C05450=1130.712,124.899,-57.710,-179.760,8.342,149.534
C05451=1130.717,124.650,-57.689,-179.762,8.338,149.533
C05452=1130.723,124.401,-57.670,-179.763,8.335,149.533
C05453=1130.727,124.152,-57.649,-179.765,8.332,149.533
C05454=1130.732,123.903,-57.630,-179.768,8.328,149.533
C05455=1130.736,123.654,-57.609,-179.770,8.325,149.532
C05456=1130.741,123.404,-57.589,-179.771,8.321,149.532
C05457=1130.746,123.156,-57.569,-179.773,8.318,149.532
C05458=1130.751,122.906,-57.550,-179.775,8.314,149.531
C05459=1130.756,122.657,-57.530,-179.777,8.311,149.531
C05460=1130.760,122.408,-57.510,-179.778,8.308,149.531
C05461=1130.765,122.159,-57.491,-179.780,8.304,149.531
C05462=1130.770,121.910,-57.470,-179.782,8.301,149.530
C05463=1130.775,121.660,-57.450,-179.784,8.297,149.530
C05464=1130.779,121.411,-57.431,-179.786,8.294,149.530
C05465=1130.784,121.162,-57.411,-179.788,8.291,149.530
C05466=1130.789,120.913,-57.391,-179.789,8.287,149.529
C05467=1130.794,120.663,-57.371,-179.791,8.284,149.529
C05468=1130.798,120.414,-57.351,-179.793,8.280,149.529
C05469=1130.804,120.166,-57.332,-179.795,8.278,149.529
C05470=1130.808,119.916,-57.312,-179.797,8.274,149.528
C05471=1130.813,119.667,-57.292,-179.799,8.271,149.528
C05472=1130.818,119.417,-57.272,-179.800,8.267,149.528
C05473=1130.823,119.169,-57.253,-179.803,8.263,149.528
C05474=1130.827,118.920,-57.233,-179.805,8.260,149.527
C05475=1130.831,118.670,-57.213,-179.806,8.257,149.527
C05476=1130.837,118.422,-57.194,-179.808,8.254,149.527
C05477=1130.841,118.172,-57.174,-179.810,8.250,149.526
C05478=1130.846,117.922,-57.155,-179.812,8.246,149.526
C05479=1130.851,117.674,-57.135,-179.814,8.243,149.526
C05480=1130.855,117.459,-57.118,-179.815,8.240,149.526
C05481=1130.859,117.244,-57.101,-179.817,8.236,149.526
C05482=1130.864,117.029,-57.084,-179.819,8.234,149.525
C05483=1130.868,116.814,-57.067,-179.820,8.231,149.525
C05484=1130.872,116.599,-57.051,-179.822,8.227,149.525
C05485=1130.877,116.384,-57.034,-179.824,8.225,149.525
C05486=1130.880,116.169,-57.017,-179.825,8.222,149.524
C05487=1130.884,115.954,-57.000,-179.827,8.219,149.524
C05488=1130.889,115.705,-56.981,-179.829,8.215,149.524
C05489=1130.894,115.456,-56.961,-179.831,8.212,149.524
C05490=1130.898,115.207,-56.941,-179.832,8.208,149.523
C05491=1130.904,114.958,-56.922,-179.834,8.205,149.523
C05492=1130.908,114.709,-56.903,-179.837,8.201,149.523
C05493=1130.913,114.460,-56.883,-179.839,8.198,149.523
C05494=1130.918,114.210,-56.864,-179.841,8.194,149.522
C05495=1130.922,113.961,-56.844,-179.843,8.191,149.522
C05496=1130.928,113.712,-56.825,-179.844,8.187,149.522
C05497=1130.932,113.463,-56.806,-179.846,8.184,149.522
C05498=1130.937,113.214,-56.786,-179.848,8.180,149.521
C05499=1130.942,112.964,-56.767,-179.851,8.177,149.521
C05500=1130.947,112.715,-56.748,-179.853,8.173,149.521
C05501=1130.951,112.466,-56.728,-179.854,8.169,149.521
C05502=1130.956,112.216,-56.709,-179.856,8.166,149.520
C05503=1130.962,111.967,-56.690,-179.858,8.162,149.520
C05504=1130.966,111.718,-56.671,-179.860,8.159,149.520
C05505=1130.971,111.469,-56.652,-179.862,8.155,149.520
C05506=1130.976,111.219,-56.632,-179.864,8.152,149.519
C05507=1130.980,110.971,-56.614,-179.866,8.148,149.519
C05508=1130.985,110.721,-56.594,-179.868,8.144,149.519
C05509=1130.990,110.472,-56.575,-179.871,8.140,149.519
C05510=1130.994,110.223,-56.556,-179.874,8.136,149.519
C05511=1131.000,109.974,-56.537,-179.877,8.132,149.518
C05512=1131.005,109.724,-56.517,-179.879,8.128,149.518
C05513=1131.009,109.475,-56.499,-179.881,8.124,149.518
C05514=1131.014,109.226,-56.479,-179.884,8.120,149.518
C05515=1131.019,108.977,-56.460,-179.887,8.117,149.518
C05516=1131.024,108.727,-56.441,-179.889,8.112,149.517
C05517=1131.029,108.478,-56.422,-179.892,8.108,149.517
C05518=1131.033,108.229,-56.403,-179.894,8.105,149.517
C05519=1131.038,107.980,-56.384,-179.897,8.100,149.517
C05520=1131.043,107.730,-56.365,-179.899,8.096,149.517
C05521=1131.048,107.481,-56.346,-179.901,8.093,149.516
C05522=1131.052,107.232,-56.327,-179.904,8.088,149.516
C05523=1131.058,106.983,-56.308,-179.907,8.084,149.516
C05524=1131.062,106.734,-56.290,-179.909,8.081,149.516
C05525=1131.067,106.484,-56.271,-179.912,8.076,149.515
C05526=1131.072,106.235,-56.252,-179.914,8.072,149.515
C05527=1131.077,105.986,-56.232,-179.916,8.068,149.515
C05528=1131.082,105.737,-56.214,-179.919,8.064,149.515
C05529=1131.086,105.487,-56.195,-179.921,8.060,149.514
C05530=1131.091,105.238,-56.177,-179.923,8.056,149.514
C05531=1131.096,104.989,-56.158,-179.925,8.052,149.514
C05532=1131.101,104.739,-56.139,-179.928,8.048,149.514
C05533=1131.106,104.491,-56.120,-179.931,8.044,149.514
C05534=1131.111,104.241,-56.102,-179.932,8.040,149.513
C05535=1131.115,103.992,-56.083,-179.935,8.036,149.513
C05536=1131.120,103.777,-56.067,-179.936,8.033,149.513
C05537=1131.123,103.562,-56.050,-179.939,8.030,149.512
C05538=1131.128,103.347,-56.034,-179.941,8.026,149.512
C05539=1131.132,103.132,-56.019,-179.943,8.023,149.512
C05540=1131.136,102.917,-56.002,-179.944,8.019,149.512
C05541=1131.140,102.702,-55.987,-179.946,8.015,149.511
C05542=1131.145,102.487,-55.970,-179.948,8.012,149.511
C05543=1131.149,102.272,-55.955,-179.950,8.008,149.511
C05544=1131.154,102.023,-55.936,-179.952,8.005,149.511
C05545=1131.158,101.773,-55.917,-179.955,8.000,149.510
C05546=1131.163,101.525,-55.898,-179.957,7.996,149.510
C05547=1131.169,101.275,-55.880,-179.958,7.993,149.510
C05548=1131.173,101.025,-55.862,-179.961,7.988,149.509
C05549=1131.178,100.776,-55.844,-179.963,7.984,149.509
C05550=1131.183,100.527,-55.825,-179.965,7.980,149.509
C05551=1131.188,100.278,-55.806,-179.967,7.976,149.508
C05552=1131.193,100.028,-55.788,-179.969,7.973,149.508
C05553=1131.197,99.780,-55.769,-179.971,7.968,149.508
C05554=1131.202,99.530,-55.751,-179.973,7.965,149.508
C05555=1131.208,99.281,-55.733,-179.976,7.960,149.507
C05556=1131.212,99.031,-55.714,-179.978,7.956,149.507
C05557=1131.217,98.782,-55.696,-179.979,7.953,149.506
C05558=1131.222,98.533,-55.678,-179.981,7.948,149.506
C05559=1131.226,98.284,-55.660,-179.983,7.944,149.506
C05560=1131.231,98.034,-55.641,-179.985,7.940,149.505
C05561=1131.236,97.785,-55.623,-179.987,7.936,149.505
C05562=1131.241,97.536,-55.605,-179.989,7.932,149.505
C05563=1131.246,97.286,-55.587,-179.991,7.928,149.504
C05564=1131.251,97.038,-55.568,-179.993,7.925,149.504
C05565=1131.255,96.788,-55.550,-179.995,7.920,149.504
C05566=1131.261,96.538,-55.531,-179.997,7.916,149.503
C05567=1131.266,96.289,-55.513,-179.998,7.912,149.503
C05568=1131.271,96.040,-55.495,180.000,7.909,149.502
C05569=1131.276,95.791,-55.477,179.997,7.904,149.502
C05570=1131.280,95.542,-55.459,179.996,7.900,149.502
C05571=1131.285,95.292,-55.441,179.994,7.896,149.501
C05572=1131.290,95.043,-55.423,179.992,7.893,149.501
C05573=1131.295,94.794,-55.405,179.990,7.888,149.500
C05574=1131.299,94.544,-55.387,179.989,7.884,149.500
C05575=1131.304,94.295,-55.369,179.987,7.881,149.500
C05576=1131.309,94.046,-55.351,179.985,7.877,149.499
C05577=1131.315,93.797,-55.332,179.983,7.873,149.499
C05578=1131.319,93.547,-55.314,179.982,7.869,149.499
C05579=1131.324,93.297,-55.296,179.980,7.864,149.498
C05580=1131.329,93.048,-55.278,179.978,7.860,149.498
C05581=1131.334,92.799,-55.260,179.976,7.856,149.497
C05582=1131.339,92.550,-55.242,179.975,7.853,149.497
C05583=1131.344,92.301,-55.224,179.973,7.849,149.496
C05584=1131.349,92.051,-55.207,179.972,7.845,149.496
C05585=1131.354,91.802,-55.189,179.970,7.841,149.496
C05586=1131.359,91.553,-55.171,179.968,7.837,149.495
C05587=1131.364,91.303,-55.153,179.967,7.833,149.495
C05588=1131.368,91.055,-55.136,179.965,7.829,149.494
C05589=1131.372,90.805,-55.117,179.964,7.825,149.494
C05590=1131.377,90.555,-55.100,179.962,7.821,149.493
C05591=1131.382,90.306,-55.082,179.960,7.817,149.493
C05592=1131.387,90.032,-55.062,179.958,7.813,149.493
C05593=1131.393,89.758,-55.043,179.957,7.809,149.492
C05594=1131.418,88.513,-54.953,-179.494,6.756,149.096
C05595=1131.423,88.264,-54.935,-179.496,6.755,149.097
C05596=1131.428,88.015,-54.918,-179.499,6.754,149.097
C05597=1131.433,87.767,-54.901,-179.502,6.753,149.098
C05598=1131.437,87.518,-54.883,-179.505,6.751,149.098
C05599=1131.443,87.268,-54.866,-179.508,6.749,149.099
C05600=1131.448,87.019,-54.848,-179.510,6.748,149.099
C05601=1131.453,86.769,-54.831,-179.513,6.746,149.100
C05602=1131.457,86.520,-54.814,-179.516,6.744,149.100
C05603=1131.462,86.271,-54.796,-179.518,6.744,149.101
C05604=1131.467,86.021,-54.778,-179.521,6.742,149.101
C05605=1131.472,85.772,-54.761,-179.524,6.740,149.101
C05606=1131.476,85.523,-54.744,-179.527,6.739,149.102
C05607=1131.482,85.273,-54.726,-179.529,6.737,149.102
C05608=1131.487,85.024,-54.708,-179.532,6.735,149.103
C05609=1131.492,84.775,-54.692,-179.535,6.734,149.103
C05610=1131.497,84.526,-54.674,-179.538,6.733,149.104
C05611=1131.502,84.276,-54.657,-179.540,6.732,149.104
C05612=1131.506,84.027,-54.640,-179.543,6.730,149.105
C05613=1131.511,83.777,-54.622,-179.546,6.728,149.105
C05614=1131.516,83.528,-54.605,-179.548,6.727,149.106
C05615=1131.521,83.278,-54.588,-179.551,6.725,149.106
C05616=1131.526,83.029,-54.570,-179.554,6.724,149.107
C05617=1131.532,82.780,-54.553,-179.557,6.723,149.107
C05618=1131.536,82.531,-54.536,-179.559,6.721,149.107
C05619=1131.541,82.281,-54.519,-179.562,6.720,149.108
C05620=1131.545,82.032,-54.502,-179.565,6.718,149.108
C05621=1131.550,81.783,-54.484,-179.568,6.716,149.109
C05622=1131.556,81.533,-54.467,-179.571,6.715,149.109
C05623=1131.561,81.284,-54.451,-179.573,6.714,149.110
C05624=1131.566,81.034,-54.433,-179.576,6.713,149.110
C05625=1131.570,80.785,-54.416,-179.578,6.711,149.111
C05626=1131.575,80.536,-54.399,-179.581,6.709,149.111
C05627=1131.580,80.286,-54.382,-179.584,6.708,149.112
C05628=1131.586,80.037,-54.365,-179.587,6.706,149.112
C05629=1131.591,79.788,-54.347,-179.589,6.705,149.113
C05630=1131.595,79.519,-54.329,-179.592,6.704,149.113
C05631=1131.601,79.251,-54.311,-179.595,6.703,149.114
C05632=1131.606,78.982,-54.293,-179.599,6.700,149.114
C05633=1131.611,78.714,-54.274,-179.601,6.698,149.115
C05634=1131.616,78.465,-54.258,-179.604,6.698,149.115
C05635=1131.621,78.215,-54.240,-179.607,6.696,149.116
C05636=1131.626,77.966,-54.224,-179.610,6.695,149.116
C05637=1131.631,77.716,-54.206,-179.612,6.693,149.116
C05638=1131.636,77.468,-54.189,-179.615,6.691,149.117
C05639=1131.641,77.218,-54.172,-179.617,6.691,149.117
C05640=1131.646,76.968,-54.155,-179.620,6.689,149.118
C05641=1131.651,76.718,-54.138,-179.623,6.688,149.118
C05642=1131.656,76.470,-54.122,-179.626,6.686,149.119
C05643=1131.661,76.220,-54.105,-179.629,6.684,149.119
C05644=1131.666,75.970,-54.088,-179.631,6.683,149.120
C05645=1131.671,75.721,-54.071,-179.634,6.682,149.120
C05646=1131.676,75.472,-54.054,-179.637,6.681,149.121
C05647=1131.680,75.222,-54.038,-179.640,6.679,149.121
C05648=1131.686,74.973,-54.020,-179.642,6.678,149.122
C05649=1131.691,74.724,-54.004,-179.644,6.676,149.122
C05650=1131.696,74.474,-53.987,-179.648,6.675,149.123
C05651=1131.700,74.225,-53.970,-179.650,6.673,149.123
C05652=1131.706,73.976,-53.954,-179.653,6.672,149.124
C05653=1131.711,73.726,-53.937,-179.655,6.671,149.124
C05654=1131.715,73.476,-53.920,-179.658,6.669,149.125
C05655=1131.720,73.228,-53.904,-179.661,6.668,149.125
C05656=1131.726,72.978,-53.886,-179.664,6.666,149.126
C05657=1131.730,72.728,-53.870,-179.666,6.666,149.126
C05658=1131.735,72.480,-53.853,-179.669,6.664,149.126
C05659=1131.740,72.230,-53.836,-179.672,6.662,149.127
C05660=1131.745,71.980,-53.819,-179.675,6.661,149.128
C05661=1131.750,71.732,-53.803,-179.678,6.659,149.128
C05662=1131.755,71.482,-53.786,-179.680,6.659,149.128
C05663=1131.760,71.232,-53.769,-179.683,6.657,149.129
C05664=1131.765,70.983,-53.754,-179.685,6.655,149.129
C05665=1131.770,70.733,-53.736,-179.689,6.654,149.130
C05666=1131.775,70.484,-53.720,-179.691,6.653,149.130
C05667=1131.780,70.235,-53.703,-179.694,6.651,149.131
C05668=1131.784,69.985,-53.687,-179.696,6.650,149.131
C05669=1131.790,69.736,-53.670,-179.699,6.648,149.132
C05670=1131.795,69.486,-53.654,-179.702,6.648,149.132
C05671=1131.800,69.237,-53.638,-179.704,6.646,149.133
C05672=1131.804,68.988,-53.621,-179.707,6.644,149.133
C05673=1131.810,68.738,-53.604,-179.709,6.644,149.134
C05674=1131.815,68.489,-53.588,-179.713,6.642,149.134
C05675=1131.819,68.239,-53.571,-179.715,6.641,149.135
C05676=1131.825,67.990,-53.555,-179.718,6.639,149.135
C05677=1131.829,67.741,-53.538,-179.720,6.638,149.136
C05678=1131.835,67.491,-53.522,-179.723,6.637,149.136
C05679=1131.840,67.242,-53.506,-179.726,6.635,149.137
C05680=1131.844,66.992,-53.489,-179.729,6.634,149.137
C05681=1131.849,66.743,-53.473,-179.731,6.633,149.138
C05682=1131.854,66.493,-53.457,-179.734,6.631,149.138
C05683=1131.859,66.245,-53.440,-179.737,6.630,149.139
C05684=1131.864,65.994,-53.424,-179.739,6.629,149.139
C05685=1131.870,65.745,-53.407,-179.742,6.627,149.140
C05686=1131.874,65.496,-53.391,-179.745,6.626,149.140
C05687=1131.880,65.246,-53.375,-179.748,6.624,149.140
C05688=1131.884,64.997,-53.359,-179.750,6.624,149.141
C05689=1131.889,64.748,-53.342,-179.753,6.622,149.142
C05690=1131.894,64.498,-53.326,-179.756,6.620,149.142
C05691=1131.899,64.249,-53.310,-179.758,6.620,149.142
C05692=1131.904,63.999,-53.294,-179.761,6.618,149.143
C05693=1131.909,63.750,-53.278,-179.764,6.617,149.143
C05694=1131.914,63.500,-53.261,-179.767,6.615,149.144
C05695=1131.919,63.251,-53.245,-179.769,6.614,149.144
C05696=1131.924,63.002,-53.228,-179.772,6.613,149.145
C05697=1131.929,62.752,-53.213,-179.775,6.611,149.145
C05698=1131.934,62.503,-53.196,-179.777,6.610,149.146
C05699=1131.939,62.253,-53.180,-179.780,6.609,149.146
C05700=1131.944,62.004,-53.164,-179.783,6.607,149.147
C05701=1131.949,61.755,-53.148,-179.785,6.607,149.147
C05702=1131.953,61.505,-53.131,-179.788,6.605,149.148
C05703=1131.959,61.256,-53.116,-179.791,6.603,149.148
C05704=1131.964,61.006,-53.100,-179.793,6.603,149.149
C05705=1131.969,60.757,-53.084,-179.796,6.601,149.149
C05706=1131.974,60.507,-53.068,-179.799,6.600,149.150
C05707=1131.979,60.258,-53.051,-179.801,6.599,149.150
C05708=1131.984,60.009,-53.036,-179.804,6.598,149.151
C05709=1131.988,59.759,-53.019,-179.807,6.596,149.151
C05710=1131.994,59.510,-53.003,-179.809,6.595,149.152
C05711=1131.999,59.260,-52.988,-179.812,6.593,149.152
C05712=1132.004,59.011,-52.971,-179.815,6.592,149.153
C05713=1132.009,58.761,-52.956,-179.817,6.591,149.153
C05714=1132.014,58.511,-52.940,-179.820,6.590,149.154
C05715=1132.018,58.263,-52.924,-179.823,6.588,149.154
C05716=1132.024,58.013,-52.908,-179.825,6.588,149.155
C05717=1132.028,57.763,-52.892,-179.828,6.586,149.155
C05718=1132.034,57.514,-52.876,-179.831,6.584,149.156
C05719=1132.038,57.264,-52.860,-179.833,6.583,149.156
C05720=1132.044,57.015,-52.845,-179.836,6.582,149.157
C05721=1132.049,56.766,-52.828,-179.839,6.581,149.157
C05722=1132.054,56.516,-52.812,-179.841,6.580,149.158
C05723=1132.059,56.267,-52.797,-179.844,6.578,149.158
C05724=1132.064,56.017,-52.781,-179.847,6.577,149.159
C05725=1132.068,55.768,-52.765,-179.849,6.576,149.159
C05726=1132.073,55.519,-52.749,-179.852,6.574,149.160
C05727=1132.079,55.269,-52.734,-179.854,6.574,149.160
C05728=1132.084,55.019,-52.718,-179.857,6.572,149.161
C05729=1132.089,54.770,-52.702,-179.860,6.571,149.161
C05730=1132.094,54.521,-52.686,-179.862,6.570,149.162
C05731=1132.099,54.271,-52.670,-179.865,6.568,149.162
C05732=1132.104,54.022,-52.655,-179.868,6.567,149.163
C05733=1132.109,53.772,-52.639,-179.871,6.566,149.163
C05734=1132.114,53.504,-52.622,-179.873,6.564,149.164
C05735=1132.120,53.235,-52.605,-179.877,6.563,149.164
C05736=1132.125,52.966,-52.588,-179.879,6.562,149.165
C05737=1132.131,52.698,-52.571,-179.883,6.560,149.166
C05738=1132.135,52.449,-52.556,-179.885,6.559,149.166
C05739=1132.141,52.199,-52.540,-179.887,6.558,149.166
C05740=1132.145,51.949,-52.525,-179.890,6.557,149.167
C05741=1132.151,51.700,-52.509,-179.893,6.556,149.168
C05742=1132.155,51.451,-52.494,-179.896,6.554,149.168
C05743=1132.161,51.201,-52.478,-179.898,6.553,149.168
C05744=1132.166,50.951,-52.462,-179.901,6.552,149.169
C05745=1132.171,50.702,-52.447,-179.903,6.551,149.170
C05746=1132.176,50.453,-52.432,-179.906,6.550,149.170
C05747=1132.181,50.203,-52.416,-179.909,6.548,149.170
C05748=1132.186,49.953,-52.400,-179.911,6.548,149.171
C05749=1132.190,49.704,-52.385,-179.914,6.546,149.172
C05750=1132.196,49.455,-52.370,-179.916,6.545,149.172
C05751=1132.201,49.205,-52.354,-179.919,6.543,149.172
C05752=1132.205,48.956,-52.339,-179.922,6.542,149.173
C05753=1132.211,48.706,-52.323,-179.924,6.541,149.174
C05754=1132.216,48.457,-52.308,-179.927,6.540,149.174
C05755=1132.221,48.208,-52.293,-179.930,6.539,149.175
C05756=1132.226,47.958,-52.277,-179.933,6.538,149.175
C05757=1132.231,47.708,-52.261,-179.935,6.537,149.176
C05758=1132.235,47.459,-52.246,-179.937,6.535,149.176
C05759=1132.241,47.210,-52.230,-179.941,6.534,149.177
C05760=1132.246,46.961,-52.215,-179.943,6.533,149.177
C05761=1132.251,46.711,-52.201,-179.946,6.531,149.178
C05762=1132.256,46.460,-52.185,-179.948,6.531,149.178
C05763=1132.261,46.211,-52.170,-179.951,6.529,149.179
C05764=1132.266,45.962,-52.154,-179.953,6.529,149.179
C05765=1132.271,45.713,-52.139,-179.956,6.527,149.180
C05766=1132.276,45.463,-52.123,-179.959,6.526,149.180
C05767=1132.281,45.214,-52.108,-179.961,6.525,149.181
C05768=1132.286,44.964,-52.094,-179.964,6.523,149.181
C05769=1132.291,44.714,-52.078,-179.967,6.523,149.182
C05770=1132.296,44.465,-52.063,-179.970,6.521,149.182
C05771=1132.301,44.216,-52.047,-179.972,6.520,149.183
C05772=1132.306,43.967,-52.032,-179.974,6.519,149.183
C05773=1132.312,43.717,-52.017,-179.977,6.518,149.184
C05774=1132.316,43.468,-52.002,-179.980,6.517,149.184
C05775=1132.322,43.218,-51.987,-179.983,6.515,149.185
C05776=1132.326,42.969,-51.972,-179.985,6.515,149.185
C05777=1132.331,42.718,-51.956,-179.988,6.513,149.186
C05778=1132.336,42.469,-51.941,-179.990,6.512,149.186
C05779=1132.341,42.220,-51.926,-179.993,6.510,149.187
C05780=1132.346,41.970,-51.912,-179.996,6.510,149.187
C05781=1132.352,41.721,-51.896,-179.998,6.508,149.188
C05782=1132.356,41.472,-51.881,179.999,6.508,149.188
C05783=1132.362,41.222,-51.866,179.996,6.506,149.189
C05784=1132.367,40.972,-51.851,179.994,6.505,149.189
C05785=1132.372,40.723,-51.836,179.991,6.504,149.190
C05786=1132.377,40.473,-51.821,179.989,6.503,149.190
C05787=1132.382,40.224,-51.806,179.986,6.502,149.191
C05788=1132.387,39.975,-51.791,179.984,6.501,149.191
C05789=1132.392,39.725,-51.776,179.981,6.499,149.192
C05790=1132.397,39.475,-51.760,179.978,6.499,149.193
C05791=1132.402,39.225,-51.746,179.976,6.497,149.193
C05792=1132.407,38.976,-51.731,179.973,6.496,149.194
C05793=1132.412,38.727,-51.716,179.971,6.495,149.194
C05794=1132.418,38.477,-51.701,179.967,6.494,149.195
C05795=1132.422,38.228,-51.686,179.965,6.493,149.195
C05796=1132.427,37.978,-51.671,179.962,6.491,149.196
C05797=1132.433,37.729,-51.656,179.960,6.491,149.196
C05798=1132.437,37.479,-51.642,179.957,6.489,149.197
C05799=1132.442,37.230,-51.627,179.955,6.488,149.197
C05800=1132.448,36.980,-51.612,179.952,6.487,149.198
C05801=1132.452,36.731,-51.597,179.949,6.486,149.198
C05802=1132.457,36.481,-51.582,179.947,6.485,149.199
C05803=1132.463,36.232,-51.567,179.944,6.484,149.199
C05804=1132.468,35.982,-51.553,179.941,6.482,149.200
C05805=1132.472,35.733,-51.538,179.939,6.482,149.200
C05806=1132.478,35.483,-51.523,179.936,6.480,149.201
C05807=1132.483,35.234,-51.508,179.934,6.480,149.201
C05808=1132.488,34.984,-51.493,179.931,6.478,149.202
C05809=1132.494,34.735,-51.479,179.929,6.477,149.202
C05810=1132.499,34.486,-51.464,179.926,6.477,149.203
C05811=1132.504,34.236,-51.450,179.923,6.475,149.203
C05812=1132.509,33.986,-51.434,179.921,6.474,149.204
C05813=1132.514,33.737,-51.420,179.918,6.473,149.205
C05814=1132.519,33.487,-51.406,179.916,6.472,149.205
C05815=1132.524,33.238,-51.391,179.913,6.471,149.205
C05816=1132.529,32.988,-51.376,179.911,6.470,149.206
C05817=1132.534,32.739,-51.361,179.908,6.469,149.207
C05818=1132.539,32.489,-51.346,179.905,6.468,149.207
C05819=1132.544,32.239,-51.332,179.903,6.466,149.207
C05820=1132.548,31.990,-51.317,179.900,6.466,149.208
C05821=1132.554,31.740,-51.302,179.897,6.464,149.209
C05822=1132.559,31.491,-51.288,179.895,6.463,149.209
C05823=1132.564,31.241,-51.274,179.892,6.462,149.210
C05824=1132.569,30.992,-51.259,179.890,6.461,149.210
C05825=1132.574,30.743,-51.245,179.887,6.460,149.211
C05826=1132.580,30.493,-51.230,179.884,6.459,149.211
C05827=1132.585,30.243,-51.216,179.882,6.458,149.212
C05828=1132.590,29.994,-51.201,179.879,6.457,149.212
C05829=1132.595,29.744,-51.186,179.877,6.456,149.213
C05830=1132.599,29.495,-51.172,179.874,6.455,149.213
C05831=1132.604,29.245,-51.158,179.872,6.454,149.214
C05832=1132.610,28.996,-51.143,179.869,6.452,149.214
C05833=1132.615,28.746,-51.128,179.866,6.452,149.215
C05834=1132.620,28.497,-51.114,179.864,6.451,149.215
C05835=1132.625,28.247,-51.100,179.861,6.449,149.216
C05836=1132.630,27.997,-51.085,179.859,6.449,149.217
C05837=1132.635,27.748,-51.071,179.856,6.447,149.217
C05838=1132.640,27.479,-51.055,179.854,6.446,149.217
C05839=1132.647,27.210,-51.040,179.851,6.445,149.218
C05840=1132.652,26.941,-51.025,179.848,6.444,149.219
C05841=1132.657,26.672,-51.009,179.845,6.443,149.219
C05842=1132.662,26.422,-50.995,179.842,6.442,149.220
C05843=1132.667,26.173,-50.980,179.840,6.441,149.220
C05844=1132.672,25.923,-50.966,179.837,6.440,149.221
C05845=1132.678,25.674,-50.952,179.835,6.439,149.221
C05846=1132.683,25.424,-50.938,179.833,6.438,149.222
C05847=1132.688,25.175,-50.924,179.829,6.437,149.222
C05848=1132.693,24.925,-50.909,179.827,6.436,149.223
C05849=1132.698,24.675,-50.895,179.824,6.434,149.223
C05850=1132.703,24.426,-50.881,179.822,6.434,149.224
C05851=1132.708,24.177,-50.866,179.820,6.433,149.225
C05852=1132.713,23.927,-50.852,179.817,6.431,149.225
C05853=1132.718,23.678,-50.838,179.814,6.431,149.226
C05854=1132.723,23.429,-50.824,179.811,6.429,149.226
C05855=1132.728,23.179,-50.809,179.809,6.428,149.227
C05856=1132.733,22.929,-50.795,179.807,6.428,149.227
C05857=1132.738,22.679,-50.782,179.804,6.426,149.228
C05858=1132.744,22.430,-50.768,179.802,6.426,149.228
C05859=1132.749,22.180,-50.753,179.798,6.424,149.229
C05860=1132.754,21.930,-50.739,179.796,6.424,149.229
C05861=1132.759,21.681,-50.725,179.794,6.423,149.230
C05862=1132.764,21.432,-50.711,179.791,6.422,149.230
C05863=1132.769,21.182,-50.697,179.789,6.421,149.231
C05864=1132.774,20.932,-50.682,179.786,6.419,149.231
C05865=1132.779,20.683,-50.668,179.783,6.419,149.232
C05866=1132.785,20.434,-50.654,179.781,6.418,149.232
C05867=1132.790,20.184,-50.640,179.778,6.416,149.233
C05868=1132.795,19.934,-50.626,179.776,6.416,149.234
C05869=1132.801,19.685,-50.612,179.773,6.415,149.234
C05870=1132.805,19.435,-50.599,179.771,6.413,149.235
C05871=1132.810,19.185,-50.584,179.768,6.413,149.235
C05872=1132.815,18.936,-50.571,179.765,6.411,149.236
C05873=1132.820,18.687,-50.556,179.763,6.411,149.236
C05874=1132.825,18.437,-50.542,179.761,6.410,149.237
C05875=1132.831,18.187,-50.529,179.758,6.409,149.237
C05876=1132.836,17.938,-50.514,179.755,6.408,149.238
C05877=1132.841,17.688,-50.500,179.753,6.407,149.238
C05878=1132.846,17.439,-50.487,179.750,6.406,149.239
C05879=1132.851,17.190,-50.473,179.748,6.405,149.239
C05880=1132.856,16.939,-50.459,179.746,6.404,149.240
C05881=1132.862,16.690,-50.445,179.742,6.403,149.240
C05882=1132.867,16.440,-50.431,179.740,6.402,149.241
C05883=1132.871,16.191,-50.417,179.737,6.400,149.241
C05884=1132.877,15.941,-50.404,179.735,6.400,149.242
C05885=1132.882,15.692,-50.390,179.733,6.399,149.243
C05886=1132.887,15.442,-50.375,179.730,6.398,149.243
C05887=1132.892,15.192,-50.362,179.727,6.397,149.244
C05888=1132.897,14.943,-50.349,179.725,6.396,149.244
C05889=1132.902,14.694,-50.335,179.722,6.395,149.245
C05890=1132.907,14.444,-50.321,179.720,6.394,149.245
C05891=1132.912,14.194,-50.307,179.717,6.393,149.246
C05892=1132.917,13.945,-50.293,179.715,6.392,149.246
C05893=1132.922,13.695,-50.280,179.712,6.391,149.247
C05894=1132.928,13.446,-50.266,179.710,6.391,149.247
C05895=1132.933,13.196,-50.252,179.707,6.389,149.248
C05896=1132.937,12.946,-50.239,179.704,6.389,149.249
C05897=1132.943,12.697,-50.225,179.702,6.388,149.249
C05898=1132.948,12.447,-50.211,179.699,6.386,149.249
C05899=1132.954,12.198,-50.197,179.697,6.386,149.250
C05900=1132.958,11.948,-50.184,179.695,6.385,149.251
C05901=1132.963,11.698,-50.170,179.692,6.383,149.251
C05902=1132.969,11.449,-50.156,179.689,6.383,149.252
C05903=1132.973,11.199,-50.143,179.687,6.382,149.252
C05904=1132.979,10.950,-50.129,179.684,6.381,149.253
C05905=1132.984,10.700,-50.116,179.682,6.380,149.253
C05906=1132.989,10.451,-50.102,179.679,6.379,149.254
C05907=1132.994,10.201,-50.089,179.677,6.378,149.254
C05908=1133.000,9.952,-50.075,179.674,6.377,149.255
C05909=1133.004,9.702,-50.062,179.672,6.376,149.255
C05910=1133.010,9.453,-50.048,179.670,6.376,149.256
C05911=1133.015,9.202,-50.035,179.666,6.374,149.257
C05912=1133.020,8.954,-50.021,179.664,6.374,149.257
C05913=1133.025,8.703,-50.008,179.662,6.373,149.257
C05914=1133.030,8.455,-49.994,179.659,6.372,149.258
C05915=1133.035,8.204,-49.981,179.657,6.371,149.259
C05916=1133.041,7.955,-49.967,179.654,6.370,149.259
C05917=1133.045,7.705,-49.954,179.652,6.370,149.260
C05918=1133.051,7.456,-49.941,179.649,6.368,149.260
C05919=1133.056,7.206,-49.927,179.647,6.367,149.261
C05920=1133.061,6.957,-49.914,179.645,6.366,149.261
C05921=1133.066,6.707,-49.900,179.641,6.365,149.262
C05922=1133.071,6.458,-49.887,179.639,6.364,149.262
C05923=1133.077,6.207,-49.873,179.637,6.364,149.263
C05924=1133.082,5.959,-49.860,179.634,6.363,149.263
C05925=1133.087,5.708,-49.847,179.632,6.361,149.264
C05926=1133.092,5.460,-49.833,179.629,6.361,149.264
C05927=1133.097,5.209,-49.820,179.627,6.360,149.265
C05928=1133.102,4.960,-49.807,179.624,6.359,149.266
C05929=1133.107,4.710,-49.793,179.622,6.358,149.266
C05930=1133.112,4.461,-49.780,179.619,6.357,149.267
C05931=1133.118,4.211,-49.767,179.617,6.357,149.267
C05932=1133.122,3.961,-49.754,179.614,6.355,149.268
C05933=1133.128,3.712,-49.740,179.612,6.355,149.268
C05934=1133.133,3.462,-49.727,179.609,6.354,149.269
C05935=1133.138,3.213,-49.714,179.607,6.353,149.269
C05936=1133.143,2.963,-49.700,179.604,6.352,149.270
C05937=1133.148,2.714,-49.687,179.602,6.351,149.270
C05938=1133.154,2.464,-49.674,179.600,6.350,149.271
C05939=1133.159,2.214,-49.661,179.597,6.350,149.272
C05940=1133.164,1.965,-49.648,179.594,6.348,149.272
C05941=1133.169,1.715,-49.634,179.592,6.347,149.272
C05942=1133.175,1.446,-49.621,179.589,6.347,149.273
C05943=1133.180,1.176,-49.606,179.587,6.345,149.274
C05944=1133.185,0.907,-49.592,179.584,6.345,149.274
C05945=1133.191,0.637,-49.578,179.581,6.343,149.275
C05946=1133.197,0.387,-49.565,179.578,6.343,149.275
C05947=1133.202,0.138,-49.552,179.576,6.342,149.276
C05948=1133.206,-0.112,-49.539,179.574,6.341,149.276
C05949=1133.212,-0.361,-49.525,179.571,6.340,149.277
C05950=1133.217,-0.611,-49.512,179.569,6.339,149.278
C05951=1133.222,-0.861,-49.499,179.566,6.339,149.278
C05952=1133.227,-1.110,-49.486,179.564,6.338,149.279
C05953=1133.232,-1.360,-49.474,179.561,6.337,149.279
C05954=1133.238,-1.610,-49.460,179.559,6.336,149.280
C05955=1133.243,-1.859,-49.448,179.556,6.335,149.280
C05956=1133.248,-2.109,-49.435,179.554,6.334,149.281
C05957=1133.253,-2.359,-49.421,179.551,6.333,149.281
C05958=1133.258,-2.608,-49.408,179.549,6.332,149.282
C05959=1133.263,-2.857,-49.395,179.546,6.332,149.282
C05960=1133.268,-3.107,-49.382,179.544,6.331,149.283
C05961=1133.274,-3.357,-49.369,179.542,6.330,149.284
C05962=1133.279,-3.606,-49.357,179.539,6.329,149.284
C05963=1133.284,-3.856,-49.344,179.537,6.328,149.285
C05964=1133.289,-4.106,-49.331,179.534,6.328,149.285
C05965=1133.294,-4.355,-49.318,179.532,6.327,149.286
C05966=1133.300,-4.604,-49.305,179.530,6.326,149.286
C05967=1133.305,-4.854,-49.292,179.526,6.325,149.287
C05968=1133.310,-5.104,-49.279,179.524,6.324,149.287
C05969=1133.315,-5.353,-49.267,179.522,6.323,149.288
C05970=1133.320,-5.603,-49.253,179.519,6.323,149.288
C05971=1133.325,-5.853,-49.240,179.517,6.322,149.289
C05972=1133.330,-6.102,-49.228,179.514,6.320,149.289
C05973=1133.336,-6.352,-49.216,179.512,6.320,149.290
C05974=1133.341,-6.602,-49.202,179.510,6.319,149.291
C05975=1133.346,-6.852,-49.190,179.507,6.318,149.291
C05976=1133.351,-7.101,-49.177,179.505,6.318,149.292
C05977=1133.356,-7.350,-49.165,179.502,6.316,149.292
C05978=1133.362,-7.601,-49.151,179.500,6.316,149.293
C05979=1133.367,-7.850,-49.138,179.497,6.315,149.293
C05980=1133.372,-8.099,-49.126,179.495,6.314,149.294
C05981=1133.377,-8.349,-49.113,179.493,6.314,149.294
C05982=1133.382,-8.598,-49.101,179.489,6.312,149.295
C05983=1133.388,-8.849,-49.088,179.487,6.312,149.295
C05984=1133.393,-9.098,-49.075,179.485,6.311,149.296
C05985=1133.398,-9.347,-49.063,179.482,6.310,149.297
C05986=1133.403,-9.597,-49.050,179.480,6.310,149.297
C05987=1133.408,-9.847,-49.037,179.478,6.309,149.298
C05988=1133.413,-10.096,-49.024,179.475,6.308,149.298
C05989=1133.418,-10.346,-49.013,179.473,6.307,149.299
C05990=1133.424,-10.596,-48.999,179.470,6.306,149.299
C05991=1133.429,-10.845,-48.987,179.468,6.306,149.300
C05992=1133.434,-11.095,-48.974,179.466,6.305,149.300
C05993=1133.439,-11.345,-48.962,179.463,6.304,149.301
C05994=1133.444,-11.594,-48.949,179.460,6.303,149.302
C05995=1133.449,-11.844,-48.937,179.458,6.302,149.302
C05996=1133.454,-12.093,-48.924,179.456,6.301,149.302
C05997=1133.460,-12.343,-48.912,179.453,6.301,149.303
C05998=1133.465,-12.593,-48.899,179.451,6.300,149.304
C05999=1133.470,-12.843,-48.886,179.449,6.299,149.304
C06000=1133.475,-13.092,-48.873,179.446,6.298,149.305
C06001=1133.481,-13.342,-48.862,179.443,6.297,149.305
C06002=1133.486,-13.591,-48.849,179.441,6.296,149.306
C06003=1133.491,-13.840,-48.836,179.439,6.296,149.306
C06004=1133.496,-14.091,-48.824,179.436,6.295,149.307
C06005=1133.501,-14.340,-48.811,179.434,6.294,149.307
C06006=1133.506,-14.590,-48.799,179.432,6.294,149.308
C06007=1133.512,-14.840,-48.787,179.429,6.293,149.309
C06008=1133.517,-15.089,-48.774,179.426,6.292,149.309
C06009=1133.522,-15.338,-48.762,179.424,6.291,149.309
C06010=1133.527,-15.588,-48.750,179.422,6.291,149.310
C06011=1133.532,-15.838,-48.737,179.419,6.290,149.311
C06012=1133.537,-16.088,-48.725,179.417,6.289,149.311
C06013=1133.542,-16.337,-48.712,179.415,6.289,149.312
C06014=1133.547,-16.587,-48.700,179.412,6.287,149.312
C06015=1133.553,-16.837,-48.688,179.410,6.286,149.313
C06016=1133.558,-17.086,-48.675,179.407,6.286,149.313
C06017=1133.563,-17.336,-48.663,179.405,6.285,149.314
C06018=1133.569,-17.585,-48.651,179.403,6.284,149.314
C06019=1133.574,-17.835,-48.639,179.400,6.284,149.315
C06020=1133.579,-18.085,-48.626,179.398,6.283,149.316
C06021=1133.584,-18.334,-48.614,179.396,6.282,149.316
C06022=1133.590,-18.584,-48.602,179.392,6.281,149.317
C06023=1133.595,-18.833,-48.589,179.390,6.280,149.317
C06024=1133.600,-19.083,-48.577,179.388,6.279,149.318
C06025=1133.605,-19.333,-48.564,179.385,6.279,149.318
C06026=1133.610,-19.583,-48.553,179.383,6.278,149.319
C06027=1133.615,-19.832,-48.540,179.381,6.277,149.319
C06028=1133.621,-20.082,-48.528,179.379,6.277,149.320
C06029=1133.626,-20.332,-48.515,179.376,6.276,149.320
C06030=1133.631,-20.582,-48.504,179.374,6.275,149.321
C06031=1133.636,-20.831,-48.492,179.371,6.274,149.321
C06032=1133.641,-21.080,-48.480,179.368,6.273,149.322
C06033=1133.646,-21.330,-48.468,179.366,6.273,149.323
C06034=1133.652,-21.580,-48.455,179.364,6.272,149.323
C06035=1133.657,-21.830,-48.443,179.361,6.271,149.324
C06036=1133.662,-22.079,-48.431,179.359,6.271,149.324
C06037=1133.668,-22.329,-48.419,179.357,6.270,149.325
C06038=1133.673,-22.579,-48.407,179.354,6.269,149.325
C06039=1133.678,-22.828,-48.394,179.352,6.269,149.326
C06040=1133.683,-23.078,-48.383,179.350,6.268,149.326
C06041=1133.688,-23.328,-48.371,179.347,6.268,149.327
C06042=1133.693,-23.577,-48.359,179.345,6.266,149.327
C06043=1133.699,-23.827,-48.347,179.342,6.265,149.328
C06044=1133.704,-24.077,-48.335,179.340,6.265,149.329
C06045=1133.709,-24.326,-48.322,179.338,6.264,149.329
C06046=1133.715,-24.596,-48.310,179.335,6.263,149.330
C06047=1133.721,-24.866,-48.297,179.333,6.263,149.330
C06048=1133.726,-25.137,-48.284,179.330,6.261,149.331
C06049=1133.732,-25.406,-48.271,179.327,6.261,149.331
C06050=1133.737,-25.656,-48.259,179.325,6.260,149.332
C06051=1133.742,-25.905,-48.247,179.323,6.259,149.332
C06052=1133.748,-26.155,-48.235,179.320,6.259,149.333
C06053=1133.752,-26.405,-48.223,179.318,6.258,149.334
C06054=1133.758,-26.655,-48.212,179.316,6.257,149.334
C06055=1133.763,-26.904,-48.199,179.313,6.257,149.335
C06056=1133.768,-27.154,-48.187,179.311,6.256,149.335
C06057=1133.773,-27.404,-48.176,179.309,6.255,149.336
C06058=1133.779,-27.654,-48.164,179.306,6.255,149.336
C06059=1133.784,-27.903,-48.151,179.304,6.254,149.337
C06060=1133.789,-28.153,-48.139,179.302,6.253,149.337
C06061=1133.794,-28.402,-48.128,179.299,6.252,149.338
C06062=1133.800,-28.652,-48.117,179.296,6.251,149.339
C06063=1133.805,-28.902,-48.105,179.294,6.251,149.339
C06064=1133.810,-29.151,-48.093,179.292,6.250,149.339
C06065=1133.815,-29.401,-48.081,179.289,6.249,149.340
C06066=1133.821,-29.651,-48.069,179.287,6.249,149.341
C06067=1133.825,-29.900,-48.058,179.285,6.248,149.341
C06068=1133.831,-30.150,-48.046,179.282,6.247,149.342
C06069=1133.836,-30.400,-48.034,179.280,6.247,149.342
C06070=1133.841,-30.650,-48.021,179.278,6.246,149.343
C06071=1133.847,-30.898,-48.010,179.275,6.245,149.343
C06072=1133.852,-31.148,-47.998,179.273,6.245,149.344
C06073=1133.857,-31.398,-47.987,179.271,6.244,149.344
C06074=1133.862,-31.648,-47.975,179.268,6.244,149.345
C06075=1133.867,-31.898,-47.963,179.266,6.243,149.346
C06076=1133.872,-32.148,-47.952,179.264,6.242,149.346
C06077=1133.878,-32.397,-47.940,179.262,6.241,149.347
C06078=1133.884,-32.647,-47.929,179.259,6.241,149.347
C06079=1133.888,-32.896,-47.917,179.257,6.240,149.348
C06080=1133.894,-33.146,-47.906,179.255,6.239,149.348
C06081=1133.899,-33.396,-47.894,179.252,6.239,149.349
C06082=1133.904,-33.646,-47.882,179.250,6.238,149.349
C06083=1133.909,-33.896,-47.870,179.248,6.237,149.350
C06084=1133.914,-34.144,-47.859,179.245,6.237,149.351
C06085=1133.920,-34.394,-47.847,179.243,6.236,149.351
C06086=1133.925,-34.644,-47.835,179.241,6.235,149.351
C06087=1133.930,-34.894,-47.824,179.238,6.235,149.352
C06088=1133.936,-35.144,-47.813,179.236,6.234,149.353
C06089=1133.941,-35.393,-47.802,179.234,6.233,149.353
C06090=1133.946,-35.643,-47.790,179.231,6.233,149.354
C06091=1133.951,-35.893,-47.778,179.229,6.232,149.354
C06092=1133.956,-36.143,-47.767,179.226,6.231,149.355
C06093=1133.961,-36.392,-47.755,179.224,6.231,149.355
C06094=1133.967,-36.641,-47.744,179.222,6.230,149.356
C06095=1133.973,-36.891,-47.732,179.219,6.229,149.356
C06096=1133.977,-37.141,-47.721,179.217,6.229,149.357
C06097=1133.983,-37.391,-47.709,179.215,6.228,149.357
C06098=1133.987,-37.641,-47.697,179.212,6.227,149.358
C06099=1133.993,-37.890,-47.686,179.210,6.227,149.359
C06100=1133.998,-38.139,-47.675,179.208,6.226,149.359
C06101=1134.004,-38.389,-47.663,179.205,6.226,149.360
C06102=1134.009,-38.640,-47.652,179.203,6.225,149.360
C06103=1134.015,-38.889,-47.641,179.201,6.224,149.361
C06104=1134.019,-39.138,-47.629,179.199,6.223,149.361
C06105=1134.025,-39.388,-47.617,179.196,6.223,149.362
C06106=1134.029,-39.638,-47.606,179.194,6.222,149.362
C06107=1134.035,-39.887,-47.595,179.192,6.221,149.363
C06108=1134.040,-40.137,-47.583,179.189,6.221,149.364
C06109=1134.046,-40.387,-47.572,179.187,6.220,149.364
C06110=1134.051,-40.636,-47.561,179.185,6.219,149.364
C06111=1134.056,-40.886,-47.550,179.183,6.219,149.365
C06112=1134.061,-41.136,-47.538,179.180,6.218,149.366
C06113=1134.066,-41.386,-47.527,179.178,6.217,149.366
C06114=1134.072,-41.635,-47.516,179.175,6.217,149.367
C06115=1134.077,-41.885,-47.505,179.173,6.216,149.367
C06116=1134.082,-42.135,-47.493,179.171,6.215,149.368
C06117=1134.088,-42.384,-47.482,179.168,6.215,149.368
C06118=1134.093,-42.634,-47.471,179.166,6.214,149.369
C06119=1134.098,-42.884,-47.459,179.164,6.213,149.369
C06120=1134.103,-43.133,-47.449,179.161,6.213,149.370
C06121=1134.109,-43.383,-47.437,179.159,6.212,149.370
C06122=1134.114,-43.633,-47.426,179.157,6.212,149.371
C06123=1134.119,-43.883,-47.415,179.154,6.211,149.372
C06124=1134.125,-44.132,-47.403,179.152,6.210,149.372
C06125=1134.130,-44.382,-47.393,179.150,6.209,149.373
C06126=1134.134,-44.632,-47.381,179.147,6.209,149.373
C06127=1134.140,-44.881,-47.370,179.145,6.208,149.374
C06128=1134.145,-45.131,-47.359,179.143,6.207,149.374
C06129=1134.151,-45.381,-47.348,179.141,6.206,149.375
C06130=1134.156,-45.630,-47.336,179.139,6.207,149.375
C06131=1134.161,-45.880,-47.326,179.136,6.206,149.376
C06132=1134.167,-46.130,-47.314,179.134,6.205,149.376
C06133=1134.172,-46.379,-47.303,179.132,6.205,149.377
C06134=1134.177,-46.630,-47.293,179.129,6.204,149.377
C06135=1134.182,-46.879,-47.282,179.127,6.203,149.378
C06136=1134.187,-47.128,-47.270,179.125,6.203,149.378
C06137=1134.192,-47.379,-47.259,179.122,6.202,149.379
C06138=1134.198,-47.628,-47.248,179.120,6.201,149.380
C06139=1134.203,-47.878,-47.237,179.118,6.201,149.380
C06140=1134.209,-48.127,-47.226,179.116,6.200,149.381
C06141=1134.213,-48.377,-47.215,179.113,6.200,149.381
C06142=1134.219,-48.627,-47.204,179.111,6.199,149.382
C06143=1134.224,-48.876,-47.193,179.109,6.198,149.382
C06144=1134.229,-49.126,-47.182,179.106,6.198,149.383
C06145=1134.235,-49.375,-47.171,179.105,6.198,149.383
C06146=1134.241,-49.626,-47.160,179.102,6.197,149.384
C06147=1134.245,-49.876,-47.149,179.100,6.196,149.384
C06148=1134.251,-50.125,-47.139,179.097,6.196,149.385
C06149=1134.255,-50.375,-47.127,179.095,6.195,149.386
C06150=1134.262,-50.645,-47.115,179.093,6.194,149.386
C06151=1134.268,-50.917,-47.104,179.090,6.194,149.387
C06152=1134.273,-51.188,-47.092,179.088,6.193,149.387
C06153=1134.279,-51.458,-47.080,179.086,6.193,149.388
C06154=1134.284,-51.707,-47.068,179.083,6.192,149.388
C06155=1134.290,-51.957,-47.058,179.081,6.191,149.389
C06156=1134.295,-52.207,-47.048,179.079,6.190,149.389
C06157=1134.299,-52.457,-47.036,179.076,6.190,149.390
C06158=1134.305,-52.706,-47.026,179.074,6.189,149.391
C06159=1134.310,-52.956,-47.015,179.072,6.188,149.391
C06160=1134.316,-53.206,-47.004,179.070,6.188,149.392
C06161=1134.321,-53.456,-46.993,179.067,6.187,149.392
C06162=1134.326,-53.705,-46.983,179.065,6.186,149.393
C06163=1134.331,-53.955,-46.972,179.063,6.186,149.393
C06164=1134.337,-54.204,-46.961,179.061,6.186,149.394
C06165=1134.342,-54.455,-46.951,179.058,6.185,149.394
C06166=1134.348,-54.704,-46.939,179.056,6.185,149.395
C06167=1134.353,-54.954,-46.928,179.054,6.184,149.395
C06168=1134.358,-55.204,-46.918,179.052,6.183,149.396
C06169=1134.363,-55.453,-46.907,179.049,6.183,149.396
C06170=1134.369,-55.703,-46.897,179.047,6.182,149.397
C06171=1134.374,-55.953,-46.886,179.045,6.181,149.397
C06172=1134.379,-56.202,-46.875,179.043,6.180,149.398
C06173=1134.384,-56.452,-46.865,179.041,6.181,149.399
C06174=1134.389,-56.702,-46.854,179.038,6.180,149.399
C06175=1134.394,-56.951,-46.843,179.036,6.179,149.400
C06176=1134.400,-57.201,-46.832,179.034,6.178,149.400
C06177=1134.405,-57.451,-46.822,179.031,6.178,149.401
C06178=1134.411,-57.700,-46.811,179.029,6.177,149.401
C06179=1134.416,-57.951,-46.800,179.027,6.177,149.402
C06180=1134.421,-58.200,-46.790,179.025,6.176,149.402
C06181=1134.426,-58.450,-46.779,179.023,6.176,149.403
C06182=1134.432,-58.699,-46.769,179.020,6.175,149.403
C06183=1134.437,-58.950,-46.758,179.018,6.175,149.404
C06184=1134.442,-59.199,-46.748,179.016,6.174,149.404
C06185=1134.447,-59.449,-46.736,179.013,6.174,149.405
C06186=1134.453,-59.698,-46.726,179.011,6.173,149.406
C06187=1134.458,-59.948,-46.716,179.009,6.172,149.406
C06188=1134.463,-60.198,-46.705,179.007,6.172,149.407
C06189=1134.469,-60.448,-46.695,179.005,6.172,149.407
C06190=1134.473,-60.697,-46.684,179.003,6.171,149.408
C06191=1134.479,-60.947,-46.674,179.000,6.170,149.408
C06192=1134.484,-61.197,-46.663,178.998,6.169,149.409
C06193=1134.490,-61.447,-46.653,178.996,6.169,149.409
C06194=1134.495,-61.697,-46.642,178.993,6.168,149.410
C06195=1134.500,-61.946,-46.631,178.992,6.168,149.410
C06196=1134.506,-62.195,-46.621,178.990,6.167,149.411
C06197=1134.511,-62.445,-46.611,178.987,6.167,149.411
C06198=1134.516,-62.695,-46.600,178.985,6.166,149.412
C06199=1134.521,-62.945,-46.590,178.982,6.166,149.412
C06200=1134.527,-63.195,-46.580,178.980,6.165,149.413
C06201=1134.532,-63.444,-46.570,178.978,6.164,149.413
C06202=1134.537,-63.694,-46.558,178.976,6.164,149.414
C06203=1134.543,-63.944,-46.548,178.974,6.164,149.415
C06204=1134.548,-64.193,-46.538,178.972,6.163,149.415
C06205=1134.553,-64.443,-46.527,178.969,6.162,149.416
C06206=1134.559,-64.693,-46.517,178.967,6.161,149.416
C06207=1134.563,-64.943,-46.507,178.965,6.161,149.417
C06208=1134.569,-65.192,-46.497,178.963,6.161,149.417
C06209=1134.574,-65.442,-46.487,178.961,6.160,149.418
C06210=1134.579,-65.692,-46.476,178.959,6.159,149.418
C06211=1134.585,-65.942,-46.466,178.956,6.159,149.419
C06212=1134.590,-66.191,-46.456,178.954,6.158,149.419
C06213=1134.595,-66.441,-46.445,178.952,6.158,149.420
C06214=1134.601,-66.691,-46.435,178.950,6.158,149.420
C06215=1134.607,-66.941,-46.425,178.948,6.157,149.421
C06216=1134.612,-67.191,-46.414,178.945,6.156,149.422
C06217=1134.616,-67.440,-46.404,178.943,6.156,149.422
C06218=1134.622,-67.690,-46.394,178.941,6.155,149.423
C06219=1134.627,-67.940,-46.384,178.939,6.155,149.423
C06220=1134.633,-68.189,-46.373,178.937,6.154,149.423
C06221=1134.638,-68.439,-46.363,178.934,6.154,149.424
C06222=1134.643,-68.689,-46.353,178.932,6.153,149.425
C06223=1134.649,-68.939,-46.342,178.930,6.152,149.425
C06224=1134.654,-69.188,-46.333,178.928,6.152,149.426
C06225=1134.659,-69.438,-46.322,178.926,6.152,149.426
C06226=1134.664,-69.688,-46.312,178.923,6.151,149.427
C06227=1134.670,-69.937,-46.302,178.921,6.150,149.427
C06228=1134.675,-70.187,-46.291,178.919,6.150,149.428
C06229=1134.680,-70.437,-46.282,178.917,6.149,149.428
C06230=1134.685,-70.686,-46.271,178.915,6.149,149.429
C06231=1134.691,-70.936,-46.261,178.913,6.149,149.429
C06232=1134.696,-71.186,-46.251,178.910,6.148,149.430
C06233=1134.702,-71.436,-46.240,178.908,6.147,149.430
C06234=1134.707,-71.685,-46.232,178.906,6.146,149.431
C06235=1134.712,-71.935,-46.221,178.904,6.147,149.432
C06236=1134.717,-72.185,-46.211,178.902,6.146,149.432
C06237=1134.723,-72.435,-46.201,178.900,6.145,149.433
C06238=1134.729,-72.684,-46.190,178.897,6.144,149.433
C06239=1134.733,-72.934,-46.181,178.896,6.144,149.434
C06240=1134.738,-73.184,-46.170,178.893,6.144,149.434
C06241=1134.744,-73.434,-46.161,178.891,6.143,149.435
C06242=1134.750,-73.683,-46.150,178.889,6.143,149.435
C06243=1134.755,-73.933,-46.141,178.887,6.142,149.436
C06244=1134.760,-74.183,-46.130,178.885,6.142,149.436
C06245=1134.765,-74.432,-46.120,178.883,6.141,149.437
C06246=1134.771,-74.683,-46.111,178.880,6.141,149.437
C06247=1134.776,-74.932,-46.101,178.878,6.140,149.438
C06248=1134.781,-75.182,-46.090,178.876,6.140,149.438
C06249=1134.787,-75.432,-46.080,178.874,6.139,149.439
C06250=1134.792,-75.681,-46.071,178.872,6.138,149.439
C06251=1134.797,-75.931,-46.061,178.869,6.138,149.440
C06252=1134.803,-76.181,-46.051,178.867,6.137,149.441
C06253=1134.808,-76.431,-46.040,178.865,6.137,149.441
C06254=1134.814,-76.702,-46.030,178.863,6.137,149.441
C06255=1134.819,-76.973,-46.020,178.861,6.136,149.442
C06256=1134.825,-77.245,-46.008,178.858,6.135,149.443
C06257=1134.831,-77.516,-45.998,178.856,6.135,149.443
C06258=1134.836,-77.766,-45.988,178.853,6.134,149.444
C06259=1134.842,-78.017,-45.978,178.851,6.134,149.444
C06260=1134.847,-78.266,-45.968,178.850,6.134,149.445
C06261=1134.853,-78.515,-45.958,178.848,6.133,149.445
C06262=1134.858,-78.765,-45.948,178.845,6.132,149.446
C06263=1134.864,-79.015,-45.939,178.843,6.131,149.446
C06264=1134.869,-79.265,-45.929,178.841,6.132,149.447
C06265=1134.873,-79.514,-45.919,178.839,6.131,149.447
C06266=1134.879,-79.764,-45.909,178.837,6.130,149.448
C06267=1134.885,-80.014,-45.899,178.834,6.129,149.448
C06268=1134.890,-80.264,-45.890,178.833,6.129,149.449
C06269=1134.896,-80.513,-45.880,178.831,6.129,149.449
C06270=1134.901,-80.764,-45.870,178.828,6.128,149.450
C06271=1134.906,-81.013,-45.861,178.826,6.128,149.451
C06272=1134.911,-81.263,-45.850,178.824,6.128,149.451
C06273=1134.916,-81.512,-45.841,178.822,6.127,149.452
C06274=1134.922,-81.762,-45.831,178.820,6.126,149.452
C06275=1134.927,-82.012,-45.822,178.818,6.125,149.453
C06276=1134.933,-82.262,-45.812,178.816,6.126,149.453
C06277=1134.938,-82.512,-45.802,178.813,6.125,149.454
C06278=1134.943,-82.761,-45.792,178.811,6.124,149.454
C06279=1134.949,-83.011,-45.783,178.810,6.124,149.455
C06280=1134.954,-83.261,-45.773,178.807,6.124,149.455
C06281=1134.959,-83.511,-45.763,178.805,6.123,149.456
C06282=1134.964,-83.760,-45.754,178.803,6.122,149.456
C06283=1134.970,-84.010,-45.744,178.801,6.122,149.457
C06284=1134.975,-84.259,-45.735,178.799,6.122,149.457
C06285=1134.981,-84.510,-45.725,178.797,6.121,149.458
C06286=1134.986,-84.759,-45.716,178.794,6.120,149.458
C06287=1134.991,-85.010,-45.706,178.793,6.120,149.459
C06288=1134.996,-85.259,-45.696,178.791,6.119,149.459
C06289=1135.002,-85.509,-45.687,178.788,6.119,149.460
C06290=1135.007,-85.758,-45.677,178.786,6.119,149.460
C06291=1135.013,-86.008,-45.668,178.784,6.118,149.461
C06292=1135.018,-86.258,-45.658,178.782,6.118,149.461
C06293=1135.023,-86.508,-45.648,178.780,6.117,149.462
C06294=1135.028,-86.757,-45.639,178.778,6.117,149.462
C06295=1135.034,-87.007,-45.629,178.776,6.116,149.463
C06296=1135.039,-87.257,-45.620,178.773,6.116,149.464
C06297=1135.045,-87.507,-45.610,178.772,6.116,149.464
C06298=1135.050,-87.756,-45.601,178.769,6.115,149.465
C06299=1135.056,-88.006,-45.591,178.767,6.114,149.465
C06300=1135.060,-88.257,-45.582,178.765,6.114,149.466
C06301=1135.065,-88.506,-45.572,178.763,6.114,149.466
C06302=1135.071,-88.756,-45.563,178.761,6.113,149.467
C06303=1135.076,-89.005,-45.553,178.759,6.113,149.467
C06304=1135.082,-89.255,-45.544,178.757,6.113,149.468
C06305=1135.087,-89.505,-45.535,178.755,6.112,149.468
C06306=1135.093,-89.755,-45.525,178.753,6.111,149.469
C06307=1135.098,-90.005,-45.516,178.751,6.111,149.469
C06308=1135.103,-90.254,-45.506,178.749,6.110,149.470
C06309=1135.109,-90.504,-45.497,178.747,6.110,149.470
C06310=1135.114,-90.754,-45.488,178.744,6.109,149.471
C06311=1135.119,-91.003,-45.477,178.742,6.109,149.471
C06312=1135.124,-91.253,-45.469,178.740,6.108,149.472
C06313=1135.130,-91.503,-45.460,178.738,6.108,149.472
C06314=1135.135,-91.753,-45.449,178.736,6.108,149.473
C06315=1135.140,-92.003,-45.441,178.734,6.107,149.473
C06316=1135.146,-92.253,-45.431,178.732,6.106,149.474
C06317=1135.151,-92.502,-45.421,178.730,6.106,149.474
C06318=1135.156,-92.752,-45.413,178.728,6.106,149.475
C06319=1135.162,-93.002,-45.403,178.726,6.105,149.475
C06320=1135.167,-93.252,-45.394,178.724,6.105,149.476
C06321=1135.172,-93.501,-45.385,178.722,6.104,149.476
C06322=1135.178,-93.751,-45.375,178.720,6.104,149.477
C06323=1135.183,-94.001,-45.366,178.718,6.104,149.477
C06324=1135.188,-94.250,-45.357,178.716,6.103,149.478
C06325=1135.194,-94.500,-45.347,178.714,6.102,149.478
C06326=1135.199,-94.750,-45.338,178.712,6.102,149.479
C06327=1135.204,-95.000,-45.329,178.710,6.102,149.479
C06328=1135.211,-95.249,-45.319,178.708,6.101,149.480
C06329=1135.216,-95.499,-45.310,178.705,6.101,149.480
C06330=1135.221,-95.749,-45.302,178.703,6.100,149.481
C06331=1135.227,-95.999,-45.292,178.701,6.100,149.481
C06332=1135.232,-96.249,-45.283,178.699,6.100,149.482
C06333=1135.237,-96.498,-45.274,178.697,6.099,149.482
C06334=1135.242,-96.748,-45.265,178.695,6.098,149.483
C06335=1135.248,-96.998,-45.255,178.694,6.098,149.483
C06336=1135.253,-97.248,-45.246,178.691,6.098,149.484
C06337=1135.258,-97.498,-45.237,178.689,6.097,149.484
C06338=1135.264,-97.747,-45.227,178.688,6.097,149.485
C06339=1135.269,-97.997,-45.218,178.685,6.096,149.486
C06340=1135.274,-98.247,-45.209,178.683,6.096,149.486
C06341=1135.279,-98.497,-45.200,178.681,6.096,149.487
C06342=1135.286,-98.746,-45.191,178.679,6.095,149.487
C06343=1135.291,-98.996,-45.182,178.677,6.094,149.488
C06344=1135.296,-99.246,-45.174,178.675,6.094,149.488
C06345=1135.301,-99.496,-45.165,178.673,6.094,149.488
C06346=1135.307,-99.745,-45.154,178.671,6.093,149.489
C06347=1135.312,-99.995,-45.146,178.669,6.093,149.489
C06348=1135.317,-100.245,-45.137,178.667,6.092,149.490
C06349=1135.322,-100.495,-45.128,178.665,6.092,149.490
C06350=1135.328,-100.745,-45.119,178.663,6.091,149.491
C06351=1135.334,-100.994,-45.110,178.660,6.091,149.492
C06352=1135.339,-101.244,-45.101,178.659,6.091,149.492
C06353=1135.344,-101.494,-45.092,178.657,6.090,149.493
C06354=1135.350,-101.744,-45.083,178.654,6.090,149.493
C06355=1135.355,-101.994,-45.074,178.653,6.090,149.494
C06356=1135.361,-102.244,-45.065,178.651,6.089,149.494
C06357=1135.366,-102.494,-45.056,178.648,6.088,149.495
C06358=1135.371,-102.766,-45.046,178.647,6.088,149.495
C06359=1135.378,-103.037,-45.036,178.645,6.087,149.496
C06360=1135.383,-103.309,-45.026,178.642,6.087,149.496
C06361=1135.389,-103.582,-45.017,178.640,6.086,149.497
C06362=1135.394,-103.832,-45.008,178.638,6.086,149.497
C06363=1135.399,-104.082,-44.999,178.636,6.086,149.498
C06364=1135.405,-104.331,-44.990,178.634,6.085,149.498
C06365=1135.411,-104.581,-44.981,178.632,6.085,149.499
C06366=1135.416,-104.831,-44.972,178.630,6.084,149.499
C06367=1135.421,-105.081,-44.963,178.628,6.084,149.500
C06368=1135.427,-105.330,-44.954,178.626,6.083,149.500
C06369=1135.432,-105.580,-44.945,178.624,6.083,149.501
C06370=1135.437,-105.830,-44.936,178.622,6.083,149.501
C06371=1135.443,-106.079,-44.928,178.620,6.082,149.502
C06372=1135.448,-106.329,-44.919,178.618,6.082,149.502
C06373=1135.453,-106.579,-44.910,178.616,6.082,149.503
C06374=1135.459,-106.830,-44.901,178.614,6.081,149.503
C06375=1135.464,-107.080,-44.892,178.612,6.081,149.504
C06376=1135.470,-107.329,-44.884,178.610,6.080,149.504
C06377=1135.475,-107.579,-44.875,178.608,6.080,149.505
C06378=1135.481,-107.828,-44.866,178.606,6.080,149.505
C06379=1135.486,-108.078,-44.857,178.604,6.079,149.506
C06380=1135.491,-108.328,-44.848,178.602,6.079,149.506
C06381=1135.497,-108.577,-44.840,178.600,6.078,149.507
C06382=1135.502,-108.827,-44.831,178.599,6.078,149.507
C06383=1135.507,-109.077,-44.822,178.596,6.077,149.508
C06384=1135.512,-109.327,-44.814,178.594,6.077,149.508
C06385=1135.518,-109.577,-44.805,178.593,6.077,149.509
C06386=1135.523,-109.826,-44.796,178.590,6.076,149.509
C06387=1135.529,-110.076,-44.787,178.589,6.076,149.510
C06388=1135.534,-110.326,-44.778,178.587,6.075,149.510
C06389=1135.539,-110.576,-44.770,178.584,6.074,149.511
C06390=1135.545,-110.825,-44.761,178.583,6.075,149.511
C06391=1135.550,-111.076,-44.753,178.581,6.074,149.512
C06392=1135.555,-111.326,-44.744,178.579,6.074,149.512
C06393=1135.560,-111.575,-44.735,178.577,6.073,149.513
C06394=1135.566,-111.824,-44.727,178.575,6.072,149.513
C06395=1135.571,-112.074,-44.718,178.573,6.072,149.514
C06396=1135.577,-112.325,-44.709,178.571,6.072,149.514
C06397=1135.583,-112.574,-44.701,178.569,6.072,149.514
C06398=1135.588,-112.824,-44.692,178.567,6.071,149.515
C06399=1135.593,-113.074,-44.683,178.565,6.070,149.515
C06400=1135.598,-113.324,-44.675,178.563,6.070,149.516
C06401=1135.604,-113.573,-44.666,178.561,6.069,149.516
C06402=1135.609,-113.823,-44.658,178.559,6.070,149.517
C06403=1135.614,-114.073,-44.649,178.557,6.069,149.517
C06404=1135.620,-114.323,-44.640,178.556,6.069,149.518
C06405=1135.626,-114.573,-44.632,178.553,6.068,149.518
C06406=1135.631,-114.822,-44.623,178.551,6.067,149.519
C06407=1135.636,-115.072,-44.614,178.550,6.067,149.519
C06408=1135.642,-115.322,-44.606,178.547,6.067,149.520
C06409=1135.647,-115.572,-44.597,178.546,6.067,149.520
C06410=1135.652,-115.822,-44.588,178.544,6.066,149.521
C06411=1135.659,-116.072,-44.581,178.542,6.066,149.521
C06412=1135.664,-116.321,-44.572,178.540,6.065,149.522
C06413=1135.669,-116.571,-44.563,178.538,6.065,149.522
C06414=1135.675,-116.821,-44.555,178.536,6.065,149.523
C06415=1135.679,-117.071,-44.547,178.534,6.064,149.523
C06416=1135.685,-117.320,-44.538,178.532,6.064,149.524
C06417=1135.691,-117.570,-44.530,178.530,6.063,149.524
C06418=1135.696,-117.820,-44.521,178.528,6.063,149.525
C06419=1135.701,-118.070,-44.512,178.526,6.062,149.525
C06420=1135.707,-118.320,-44.504,178.525,6.062,149.526
C06421=1135.712,-118.570,-44.496,178.522,6.062,149.526
C06422=1135.717,-118.819,-44.487,178.521,6.062,149.527
C06423=1135.723,-119.069,-44.479,178.519,6.061,149.527
C06424=1135.728,-119.319,-44.471,178.516,6.060,149.528
C06425=1135.733,-119.569,-44.462,178.515,6.060,149.528
C06426=1135.739,-119.818,-44.454,178.513,6.060,149.529
C06427=1135.744,-120.068,-44.445,178.511,6.060,149.529
C06428=1135.750,-120.319,-44.437,178.509,6.059,149.530
C06429=1135.756,-120.568,-44.428,178.507,6.059,149.530
C06430=1135.760,-120.818,-44.421,178.505,6.058,149.531
C06431=1135.766,-121.067,-44.412,178.503,6.058,149.531
C06432=1135.771,-121.317,-44.403,178.501,6.057,149.532
C06433=1135.777,-121.567,-44.395,178.500,6.058,149.532
C06434=1135.782,-121.817,-44.386,178.497,6.057,149.533
C06435=1135.788,-122.067,-44.378,178.495,6.056,149.533
C06436=1135.792,-122.317,-44.370,178.494,6.056,149.533
C06437=1135.798,-122.566,-44.362,178.491,6.055,149.534
C06438=1135.804,-122.816,-44.353,178.490,6.055,149.534
C06439=1135.810,-123.066,-44.345,178.488,6.055,149.535
C06440=1135.815,-123.316,-44.337,178.486,6.055,149.535
C06441=1135.820,-123.566,-44.329,178.484,6.054,149.536
C06442=1135.825,-123.815,-44.320,178.482,6.054,149.536
C06443=1135.831,-124.066,-44.312,178.480,6.053,149.537
C06444=1135.837,-124.315,-44.304,178.479,6.053,149.537
C06445=1135.841,-124.565,-44.296,178.476,6.053,149.538
C06446=1135.847,-124.814,-44.288,178.475,6.052,149.538
C06447=1135.853,-125.065,-44.279,178.473,6.051,149.539
C06448=1135.858,-125.314,-44.271,178.471,6.052,149.539
C06449=1135.863,-125.564,-44.263,178.469,6.051,149.540
C06450=1135.868,-125.814,-44.254,178.468,6.051,149.540
C06451=1135.874,-126.063,-44.247,178.465,6.050,149.541
C06452=1135.879,-126.313,-44.238,178.464,6.050,149.541
C06453=1135.885,-126.563,-44.230,178.462,6.049,149.542
C06454=1135.890,-126.813,-44.222,178.459,6.049,149.542
C06455=1135.895,-127.063,-44.213,178.458,6.049,149.543
C06456=1135.901,-127.313,-44.206,178.456,6.048,149.543
C06457=1135.906,-127.562,-44.197,178.454,6.048,149.544
C06458=1135.912,-127.812,-44.189,178.452,6.047,149.544
C06459=1135.917,-128.062,-44.181,178.450,6.047,149.544
C06460=1135.922,-128.311,-44.173,178.448,6.047,149.545
C06461=1135.928,-128.562,-44.165,178.447,6.046,149.545
C06462=1135.508,-128.573,-44.209,178.443,6.050,149.547
C06463=1135.502,-128.323,-44.217,178.445,6.050,149.547
C06464=1135.496,-128.073,-44.225,178.447,6.050,149.546
C06465=1135.491,-127.823,-44.234,178.449,6.051,149.546
C06466=1135.486,-127.574,-44.241,178.451,6.051,149.545
C06467=1135.480,-127.324,-44.250,178.452,6.052,149.545
C06468=1135.474,-127.074,-44.257,178.455,6.053,149.544
C06469=1135.469,-126.824,-44.266,178.456,6.053,149.544
C06470=1135.464,-126.575,-44.274,178.458,6.053,149.543
C06471=1135.458,-126.324,-44.282,178.460,6.053,149.543
C06472=1135.453,-126.075,-44.291,178.462,6.054,149.542
C06473=1135.448,-125.825,-44.298,178.464,6.054,149.542
C06474=1135.443,-125.575,-44.307,178.466,6.055,149.541
C06475=1135.437,-125.325,-44.315,178.468,6.055,149.541
C06476=1135.431,-125.076,-44.324,178.470,6.056,149.540
C06477=1135.426,-124.826,-44.331,178.471,6.056,149.540
C06478=1135.421,-124.576,-44.340,178.474,6.056,149.539
C06479=1135.415,-124.326,-44.348,178.475,6.056,149.539
C06480=1135.409,-124.076,-44.356,178.477,6.057,149.538
C06481=1135.404,-123.826,-44.365,178.479,6.057,149.538
C06482=1135.399,-123.577,-44.372,178.481,6.058,149.538
C06483=1135.394,-123.327,-44.381,178.483,6.058,149.537
C06484=1135.389,-123.077,-44.390,178.484,6.059,149.537
C06485=1135.382,-122.827,-44.397,178.486,6.059,149.536
C06486=1135.378,-122.578,-44.406,178.488,6.059,149.536
C06487=1135.372,-122.328,-44.413,178.490,6.059,149.535
C06488=1135.367,-122.078,-44.422,178.492,6.060,149.535
C06489=1135.361,-121.828,-44.431,178.494,6.061,149.534
C06490=1135.356,-121.579,-44.439,178.496,6.061,149.534
C06491=1135.351,-121.328,-44.447,178.498,6.062,149.533
C06492=1135.345,-121.079,-44.455,178.500,6.062,149.533
C06493=1135.340,-120.829,-44.463,178.502,6.062,149.532
C06494=1135.334,-120.579,-44.472,178.503,6.062,149.532
C06495=1135.329,-120.330,-44.481,178.506,6.063,149.531
C06496=1135.323,-120.079,-44.489,178.507,6.063,149.531
C06497=1135.319,-119.830,-44.497,178.509,6.064,149.530
C06498=1135.313,-119.580,-44.505,178.511,6.064,149.530
C06499=1135.308,-119.330,-44.514,178.513,6.064,149.529
C06500=1135.302,-119.080,-44.523,178.515,6.065,149.529
C06501=1135.296,-118.830,-44.531,178.517,6.065,149.528
C06502=1135.291,-118.581,-44.540,178.519,6.066,149.528
C06503=1135.286,-118.330,-44.548,178.521,6.066,149.528
C06504=1135.280,-118.081,-44.556,178.523,6.066,149.527
C06505=1135.275,-117.831,-44.565,178.525,6.066,149.527
C06506=1135.269,-117.582,-44.572,178.527,6.067,149.526
C06507=1135.264,-117.332,-44.581,178.528,6.067,149.526
C06508=1135.259,-117.082,-44.590,178.531,6.068,149.525
C06509=1135.253,-116.832,-44.598,178.533,6.069,149.525
C06510=1135.248,-116.582,-44.607,178.534,6.069,149.524
C06511=1135.243,-116.333,-44.616,178.537,6.069,149.524
C06512=1135.237,-116.082,-44.624,178.538,6.069,149.523
C06513=1135.231,-115.833,-44.633,178.540,6.070,149.523
C06514=1135.226,-115.583,-44.642,178.542,6.070,149.522
C06515=1135.221,-115.333,-44.650,178.544,6.071,149.522
C06516=1135.215,-115.083,-44.658,178.546,6.071,149.521
C06517=1135.211,-114.834,-44.667,178.548,6.071,149.521
C06518=1135.205,-114.584,-44.675,178.550,6.072,149.520
C06519=1135.199,-114.334,-44.683,178.552,6.072,149.520
C06520=1135.194,-114.084,-44.692,178.554,6.073,149.519
C06521=1135.189,-113.835,-44.701,178.556,6.073,149.519
C06522=1135.183,-113.585,-44.710,178.558,6.074,149.518
C06523=1135.178,-113.335,-44.718,178.559,6.074,149.518
C06524=1135.173,-113.085,-44.727,178.562,6.074,149.517
C06525=1135.167,-112.835,-44.736,178.564,6.075,149.517
C06526=1135.162,-112.586,-44.744,178.565,6.075,149.516
C06527=1135.156,-112.336,-44.752,178.568,6.076,149.516
C06528=1135.151,-112.086,-44.761,178.569,6.076,149.515
C06529=1135.146,-111.836,-44.770,178.571,6.076,149.515
C06530=1135.140,-111.587,-44.779,178.574,6.077,149.514
C06531=1135.135,-111.337,-44.787,178.575,6.077,149.514
C06532=1135.129,-111.086,-44.796,178.577,6.078,149.513
C06533=1135.124,-110.837,-44.804,178.579,6.078,149.513
C06534=1135.119,-110.587,-44.813,178.581,6.079,149.512
C06535=1135.113,-110.338,-44.822,178.583,6.079,149.512
C06536=1135.108,-110.088,-44.831,178.585,6.079,149.511
C06537=1135.103,-109.838,-44.840,178.587,6.080,149.511
C06538=1135.097,-109.588,-44.848,178.589,6.080,149.510
C06539=1135.092,-109.338,-44.857,178.591,6.081,149.510
C06540=1135.087,-109.088,-44.865,178.593,6.081,149.509
C06541=1135.081,-108.839,-44.874,178.595,6.081,149.509
C06542=1135.076,-108.589,-44.883,178.597,6.082,149.508
C06543=1135.070,-108.339,-44.892,178.599,6.082,149.508
C06544=1135.065,-108.089,-44.901,178.601,6.083,149.508
C06545=1135.059,-107.840,-44.910,178.602,6.083,149.507
C06546=1135.054,-107.589,-44.918,178.604,6.084,149.507
C06547=1135.048,-107.340,-44.927,178.607,6.084,149.506
C06548=1135.043,-107.090,-44.936,178.608,6.084,149.506
C06549=1135.038,-106.840,-44.945,178.610,6.085,149.505
C06550=1135.033,-106.590,-44.954,178.613,6.086,149.505
C06551=1135.028,-106.341,-44.962,178.614,6.086,149.504
C06552=1135.022,-106.091,-44.971,178.616,6.086,149.504
C06553=1135.017,-105.842,-44.980,178.618,6.086,149.503
C06554=1135.011,-105.592,-44.989,178.621,6.087,149.502
C06555=1135.006,-105.342,-44.998,178.623,6.088,149.502
C06556=1135.000,-105.092,-45.007,178.625,6.087,149.501
C06557=1134.995,-104.843,-45.016,178.627,6.088,149.501
C06558=1134.989,-104.593,-45.025,178.628,6.088,149.501
C06559=1134.984,-104.343,-45.033,178.631,6.089,149.500
C06560=1134.979,-104.093,-45.042,178.633,6.090,149.500
C06561=1134.974,-103.843,-45.051,178.634,6.090,149.499
C06562=1134.969,-103.593,-45.060,178.637,6.090,149.499
C06563=1134.962,-103.321,-45.069,178.639,6.091,149.498
C06564=1134.956,-103.049,-45.079,178.640,6.091,149.498
C06565=1134.950,-102.777,-45.090,178.643,6.091,149.497
C06566=1134.945,-102.504,-45.099,178.645,6.092,149.496
C06567=1134.939,-102.254,-45.108,178.647,6.093,149.496
C06568=1134.934,-102.004,-45.117,178.649,6.093,149.495
C06569=1134.929,-101.755,-45.126,178.651,6.094,149.495
C06570=1134.924,-101.505,-45.135,178.653,6.094,149.494
C06571=1134.917,-101.255,-45.144,178.655,6.094,149.494
C06572=1134.912,-101.005,-45.153,178.657,6.095,149.493
C06573=1134.907,-100.756,-45.162,178.659,6.095,149.493
C06574=1134.902,-100.506,-45.171,178.661,6.095,149.492
C06575=1134.897,-100.256,-45.180,178.664,6.096,149.492
C06576=1134.891,-100.006,-45.190,178.665,6.096,149.491
C06577=1134.886,-99.756,-45.199,178.667,6.097,149.491
C06578=1134.881,-99.507,-45.207,178.670,6.098,149.490
C06579=1134.875,-99.257,-45.216,178.671,6.098,149.490
C06580=1134.869,-99.007,-45.226,178.673,6.098,149.489
C06581=1134.864,-98.757,-45.234,178.676,6.099,149.489
C06582=1134.859,-98.508,-45.244,178.677,6.099,149.488
C06583=1134.854,-98.258,-45.253,178.679,6.100,149.488
C06584=1134.848,-98.008,-45.262,178.682,6.101,149.487
C06585=1134.843,-97.758,-45.271,178.683,6.100,149.487
C06586=1134.838,-97.508,-45.280,178.685,6.101,149.486
C06587=1134.832,-97.259,-45.289,178.688,6.102,149.486
C06588=1134.827,-97.008,-45.299,178.690,6.102,149.485
C06589=1134.822,-96.759,-45.308,178.692,6.102,149.485
C06590=1134.816,-96.510,-45.317,178.694,6.103,149.484
C06591=1134.810,-96.260,-45.326,178.696,6.103,149.484
C06592=1134.805,-96.010,-45.335,178.698,6.104,149.483
C06593=1134.800,-95.760,-45.344,178.700,6.105,149.483
C06594=1134.795,-95.511,-45.354,178.702,6.104,149.482
C06595=1134.789,-95.261,-45.363,178.704,6.105,149.482
C06596=1134.784,-95.011,-45.372,178.706,6.106,149.481
C06597=1134.779,-94.761,-45.381,178.708,6.106,149.481
C06598=1134.773,-94.512,-45.391,178.710,6.106,149.480
C06599=1134.768,-94.262,-45.400,178.713,6.107,149.480
C06600=1134.763,-94.012,-45.409,178.714,6.107,149.479
C06601=1134.757,-93.762,-45.418,178.716,6.108,149.479
C06602=1134.752,-93.512,-45.428,178.718,6.109,149.478
C06603=1134.747,-93.263,-45.437,178.720,6.108,149.478
C06604=1134.741,-93.012,-45.446,178.722,6.109,149.477
C06605=1134.736,-92.763,-45.456,178.724,6.110,149.477
C06606=1134.731,-92.513,-45.465,178.726,6.110,149.476
C06607=1134.725,-92.263,-45.474,178.729,6.110,149.476
C06608=1134.720,-92.013,-45.483,178.731,6.111,149.475
C06609=1134.714,-91.764,-45.494,178.733,6.111,149.475
C06610=1134.709,-91.514,-45.502,178.735,6.112,149.474
C06611=1134.704,-91.264,-45.511,178.737,6.113,149.474
C06612=1134.698,-91.015,-45.522,178.739,6.113,149.473
C06613=1134.693,-90.765,-45.530,178.741,6.113,149.473
C06614=1134.688,-90.515,-45.539,178.743,6.114,149.472
C06615=1134.682,-90.265,-45.550,178.745,6.114,149.471
C06616=1134.677,-90.015,-45.558,178.747,6.114,149.471
C06617=1134.672,-89.766,-45.569,178.749,6.115,149.470
C06618=1134.666,-89.516,-45.578,178.752,6.116,149.470
C06619=1134.660,-89.266,-45.587,178.753,6.116,149.470
C06620=1134.656,-89.017,-45.597,178.755,6.117,149.469
C06621=1134.650,-88.767,-45.606,178.758,6.117,149.469
C06622=1134.645,-88.517,-45.615,178.759,6.117,149.468
C06623=1134.640,-88.267,-45.625,178.762,6.118,149.467
C06624=1134.634,-88.017,-45.634,178.764,6.118,149.467
C06625=1134.629,-87.768,-45.644,178.766,6.119,149.466
C06626=1134.623,-87.518,-45.653,178.768,6.119,149.466
C06627=1134.618,-87.269,-45.663,178.770,6.120,149.465
C06628=1134.613,-87.019,-45.672,178.772,6.121,149.465
C06629=1134.607,-86.769,-45.682,178.774,6.121,149.464
C06630=1134.603,-86.519,-45.691,178.776,6.121,149.464
C06631=1134.597,-86.269,-45.701,178.779,6.122,149.463
C06632=1134.592,-86.019,-45.710,178.780,6.122,149.463
C06633=1134.586,-85.769,-45.720,178.782,6.122,149.462
C06634=1134.581,-85.520,-45.729,178.785,6.123,149.462
C06635=1134.575,-85.270,-45.739,178.787,6.124,149.461
C06636=1134.571,-85.021,-45.749,178.788,6.124,149.461
C06637=1134.565,-84.770,-45.758,178.791,6.125,149.460
C06638=1134.560,-84.521,-45.768,178.793,6.125,149.460
C06639=1134.554,-84.271,-45.777,178.796,6.126,149.459
C06640=1134.549,-84.022,-45.787,178.797,6.126,149.459
C06641=1134.544,-83.771,-45.797,178.799,6.126,149.458
C06642=1134.539,-83.522,-45.806,178.801,6.127,149.458
C06643=1134.533,-83.272,-45.816,178.803,6.127,149.457
C06644=1134.527,-83.022,-45.826,178.805,6.128,149.457
C06645=1134.522,-82.773,-45.836,178.808,6.128,149.456
C06646=1134.517,-82.523,-45.845,178.810,6.129,149.456
C06647=1134.512,-82.273,-45.855,178.812,6.129,149.455
C06648=1134.506,-82.023,-45.864,178.814,6.130,149.455
C06649=1134.501,-81.774,-45.874,178.816,6.131,149.454
C06650=1134.496,-81.524,-45.884,178.818,6.131,149.454
C06651=1134.490,-81.273,-45.894,178.820,6.131,149.453
C06652=1134.485,-81.024,-45.903,178.823,6.132,149.452
C06653=1134.479,-80.774,-45.913,178.825,6.132,149.452
C06654=1134.474,-80.525,-45.923,178.827,6.133,149.451
C06655=1134.469,-80.275,-45.933,178.829,6.133,149.451
C06656=1134.463,-80.025,-45.942,178.831,6.134,149.450
C06657=1134.459,-79.775,-45.952,178.833,6.134,149.450
C06658=1134.453,-79.526,-45.962,178.836,6.135,149.449
C06659=1134.448,-79.276,-45.971,178.837,6.135,149.449
C06660=1134.442,-79.026,-45.982,178.839,6.136,149.448
C06661=1134.437,-78.777,-45.992,178.842,6.137,149.448
C06662=1134.432,-78.527,-46.001,178.844,6.137,149.447
C06663=1134.427,-78.277,-46.011,178.846,6.137,149.447
C06664=1134.421,-78.027,-46.021,178.848,6.138,149.446
C06665=1134.416,-77.777,-46.030,178.850,6.138,149.446
C06666=1134.410,-77.528,-46.041,178.852,6.139,149.445
C06667=1134.405,-77.256,-46.052,178.855,6.140,149.445
C06668=1134.398,-76.985,-46.062,178.857,6.139,149.444
C06669=1134.393,-76.714,-46.073,178.859,6.140,149.444
C06670=1134.387,-76.441,-46.084,178.861,6.141,149.443
C06671=1134.382,-76.192,-46.093,178.864,6.141,149.442
C06672=1134.376,-75.943,-46.104,178.866,6.142,149.442
C06673=1134.371,-75.692,-46.114,178.868,6.143,149.441
C06674=1134.366,-75.442,-46.123,178.870,6.143,149.441
C06675=1134.360,-75.193,-46.133,178.872,6.144,149.440
C06676=1134.355,-74.943,-46.143,178.875,6.144,149.440
C06677=1134.349,-74.694,-46.154,178.877,6.145,149.439
C06678=1134.345,-74.443,-46.163,178.879,6.145,149.439
C06679=1134.339,-74.194,-46.173,178.881,6.145,149.438
C06680=1134.334,-73.944,-46.183,178.883,6.146,149.438
C06681=1134.328,-73.695,-46.194,178.885,6.147,149.437
C06682=1134.324,-73.445,-46.204,178.888,6.147,149.437
C06683=1134.318,-73.195,-46.213,178.889,6.147,149.436
C06684=1134.312,-72.945,-46.223,178.891,6.148,149.436
C06685=1134.307,-72.695,-46.233,178.894,6.149,149.435
C06686=1134.302,-72.446,-46.243,178.896,6.150,149.435
C06687=1134.297,-72.196,-46.254,178.899,6.150,149.434
C06688=1134.291,-71.946,-46.264,178.900,6.150,149.433
C06689=1134.286,-71.697,-46.274,178.902,6.151,149.433
C06690=1134.281,-71.446,-46.283,178.904,6.151,149.432
C06691=1134.275,-71.197,-46.293,178.907,6.152,149.432
C06692=1134.270,-70.947,-46.304,178.909,6.153,149.431
C06693=1134.264,-70.698,-46.314,178.911,6.153,149.431
C06694=1134.259,-70.447,-46.324,178.913,6.153,149.430
C06695=1134.254,-70.198,-46.334,178.915,6.154,149.430
C06696=1134.249,-69.949,-46.344,178.918,6.155,149.429
C06697=1134.244,-69.698,-46.355,178.920,6.155,149.429
C06698=1134.238,-69.449,-46.365,178.922,6.155,149.428
C06699=1134.233,-69.199,-46.375,178.924,6.156,149.428
C06700=1134.227,-68.950,-46.386,178.926,6.157,149.427
C06701=1134.223,-68.700,-46.395,178.928,6.157,149.427
C06702=1134.217,-68.450,-46.406,178.931,6.158,149.426
C06703=1134.211,-68.201,-46.416,178.933,6.158,149.426
C06704=1134.206,-67.951,-46.426,178.935,6.159,149.425
C06705=1134.201,-67.701,-46.437,178.937,6.159,149.425
C06706=1134.195,-67.452,-46.447,178.939,6.160,149.424
C06707=1134.190,-67.201,-46.457,178.942,6.160,149.423
C06708=1134.185,-66.952,-46.467,178.944,6.161,149.423
C06709=1134.180,-66.702,-46.477,178.946,6.161,149.422
C06710=1134.175,-66.452,-46.488,178.948,6.162,149.422
C06711=1134.169,-66.203,-46.498,178.951,6.162,149.421
C06712=1134.164,-65.953,-46.508,178.953,6.163,149.421
C06713=1134.159,-65.703,-46.519,178.955,6.164,149.420
C06714=1134.153,-65.453,-46.529,178.957,6.165,149.420
C06715=1134.147,-65.204,-46.539,178.959,6.165,149.419
C06716=1134.142,-64.954,-46.550,178.961,6.165,149.419
C06717=1134.137,-64.704,-46.560,178.964,6.166,149.418
C06718=1134.133,-64.454,-46.570,178.966,6.167,149.418
C06719=1134.127,-64.205,-46.580,178.968,6.167,149.417
C06720=1134.121,-63.955,-46.590,178.970,6.168,149.417
C06721=1134.116,-63.705,-46.601,178.972,6.168,149.416
C06722=1134.111,-63.455,-46.611,178.974,6.168,149.415
C06723=1134.105,-63.206,-46.622,178.977,6.169,149.415
C06724=1134.100,-62.956,-46.633,178.979,6.170,149.415
C06725=1134.095,-62.707,-46.643,178.981,6.170,149.414
C06726=1134.090,-62.456,-46.654,178.984,6.171,149.413
C06727=1134.084,-62.207,-46.664,178.985,6.171,149.413
C06728=1134.079,-61.957,-46.674,178.987,6.172,149.412
C06729=1134.074,-61.707,-46.685,178.990,6.173,149.412
C06730=1134.068,-61.458,-46.695,178.992,6.173,149.411
C06731=1134.063,-61.208,-46.706,178.994,6.174,149.411
C06732=1134.058,-60.958,-46.716,178.997,6.174,149.410
C06733=1134.053,-60.708,-46.727,178.999,6.175,149.410
C06734=1134.047,-60.458,-46.737,179.001,6.175,149.409
C06735=1134.042,-60.210,-46.748,179.003,6.176,149.409
C06736=1134.037,-59.959,-46.759,179.005,6.176,149.408
C06737=1134.031,-59.710,-46.769,179.008,6.177,149.408
C06738=1134.026,-59.459,-46.779,179.010,6.177,149.407
C06739=1134.021,-59.211,-46.790,179.012,6.178,149.406
C06740=1134.016,-58.960,-46.801,179.015,6.179,149.406
C06741=1134.010,-58.711,-46.811,179.016,6.179,149.405
C06742=1134.005,-58.461,-46.822,179.018,6.180,149.405
C06743=1134.000,-58.212,-46.832,179.021,6.180,149.404
C06744=1133.995,-57.961,-46.843,179.023,6.181,149.404
C06745=1133.990,-57.712,-46.853,179.025,6.182,149.403
C06746=1133.985,-57.462,-46.864,179.028,6.182,149.403
C06747=1133.979,-57.213,-46.875,179.030,6.183,149.402
C06748=1133.974,-56.963,-46.885,179.032,6.184,149.402
C06749=1133.968,-56.713,-46.896,179.034,6.184,149.401
C06750=1133.963,-56.464,-46.907,179.036,6.184,149.401
C06751=1133.958,-56.213,-46.918,179.039,6.185,149.400
C06752=1133.952,-55.964,-46.928,179.041,6.186,149.399
C06753=1133.947,-55.714,-46.939,179.043,6.186,149.399
C06754=1133.942,-55.465,-46.949,179.045,6.187,149.399
C06755=1133.937,-55.214,-46.960,179.048,6.187,149.398
C06756=1133.932,-54.965,-46.971,179.050,6.188,149.397
C06757=1133.926,-54.715,-46.981,179.053,6.189,149.397
C06758=1133.922,-54.466,-46.993,179.054,6.189,149.396
C06759=1133.915,-54.216,-47.004,179.057,6.189,149.396
C06760=1133.910,-53.966,-47.014,179.059,6.190,149.395
C06761=1133.905,-53.717,-47.025,179.061,6.191,149.395
C06762=1133.900,-53.466,-47.036,179.063,6.192,149.394
C06763=1133.895,-53.217,-47.047,179.066,6.192,149.394
C06764=1133.890,-52.967,-47.057,179.068,6.193,149.393
C06765=1133.884,-52.717,-47.068,179.070,6.194,149.393
C06766=1133.879,-52.468,-47.079,179.073,6.194,149.392
C06767=1133.873,-52.218,-47.089,179.075,6.195,149.391
C06768=1133.869,-51.969,-47.101,179.077,6.195,149.391
C06769=1133.863,-51.719,-47.111,179.079,6.195,149.390
C06770=1133.857,-51.469,-47.123,179.081,6.196,149.390
C06771=1133.852,-51.198,-47.134,179.084,6.197,149.389
C06772=1133.846,-50.927,-47.146,179.086,6.197,149.389
C06773=1133.840,-50.657,-47.158,179.089,6.199,149.388
C06774=1133.835,-50.386,-47.170,179.092,6.199,149.388
C06775=1133.829,-50.136,-47.180,179.094,6.200,149.387
C06776=1133.825,-49.886,-47.192,179.096,6.200,149.386
C06777=1133.819,-49.637,-47.202,179.098,6.200,149.386
C06778=1133.814,-49.387,-47.214,179.100,6.201,149.385
C06779=1133.808,-49.137,-47.224,179.103,6.202,149.385
C06780=1133.803,-48.888,-47.235,179.105,6.202,149.384
C06781=1133.799,-48.638,-47.246,179.107,6.203,149.384
C06782=1133.792,-48.388,-47.257,179.109,6.204,149.383
C06783=1133.788,-48.139,-47.269,179.112,6.204,149.383
C06784=1133.782,-47.889,-47.279,179.114,6.205,149.382
C06785=1133.777,-47.639,-47.290,179.116,6.206,149.382
C06786=1133.772,-47.389,-47.301,179.119,6.207,149.381
C06787=1133.766,-47.140,-47.312,179.121,6.207,149.380
C06788=1133.762,-46.890,-47.323,179.124,6.208,149.380
C06789=1133.756,-46.640,-47.335,179.126,6.209,149.380
C06790=1133.750,-46.391,-47.346,179.128,6.209,149.379
C06791=1133.746,-46.141,-47.357,179.130,6.209,149.378
C06792=1133.740,-45.891,-47.368,179.132,6.210,149.378
C06793=1133.735,-45.642,-47.379,179.134,6.210,149.377
C06794=1133.730,-45.391,-47.390,179.137,6.211,149.377
C06795=1133.724,-45.142,-47.401,179.139,6.212,149.376
C06796=1133.719,-44.893,-47.412,179.141,6.212,149.376
C06797=1133.714,-44.642,-47.423,179.144,6.213,149.375
C06798=1133.708,-44.393,-47.434,179.146,6.214,149.375
C06799=1133.703,-44.144,-47.446,179.148,6.214,149.374
C06800=1133.699,-43.894,-47.457,179.151,6.215,149.374
C06801=1133.692,-43.644,-47.468,179.153,6.216,149.373
C06802=1133.688,-43.394,-47.479,179.155,6.216,149.372
C06803=1133.682,-43.144,-47.491,179.158,6.217,149.372
C06804=1133.677,-42.895,-47.501,179.160,6.218,149.371
C06805=1133.672,-42.645,-47.512,179.163,6.218,149.371
C06806=1133.666,-42.395,-47.524,179.165,6.219,149.370
C06807=1133.662,-42.146,-47.536,179.167,6.220,149.370
C06808=1133.655,-41.896,-47.546,179.169,6.221,149.369
C06809=1133.651,-41.646,-47.558,179.172,6.221,149.369
C06810=1133.646,-41.397,-47.569,179.174,6.222,149.368
C06811=1133.640,-41.147,-47.581,179.176,6.223,149.368
C06812=1133.635,-40.898,-47.592,179.178,6.223,149.367
C06813=1133.630,-40.647,-47.603,179.181,6.224,149.366
C06814=1133.625,-40.398,-47.614,179.183,6.224,149.366
C06815=1133.619,-40.148,-47.626,179.185,6.225,149.366
C06816=1133.614,-39.899,-47.637,179.188,6.226,149.365
C06817=1133.609,-39.649,-47.649,179.190,6.226,149.364
C06818=1133.603,-39.399,-47.659,179.192,6.227,149.364
C06819=1133.598,-39.149,-47.671,179.195,6.228,149.363
C06820=1133.593,-38.900,-47.682,179.197,6.228,149.363
C06821=1133.588,-38.650,-47.694,179.199,6.229,149.362
C06822=1133.582,-38.401,-47.705,179.202,6.230,149.362
C06823=1133.577,-38.151,-47.717,179.204,6.230,149.361
C06824=1133.572,-37.901,-47.728,179.206,6.230,149.361
C06825=1133.567,-37.651,-47.740,179.208,6.231,149.360
C06826=1133.561,-37.402,-47.750,179.210,6.232,149.360
C06827=1133.556,-37.152,-47.762,179.213,6.232,149.359
C06828=1133.551,-36.902,-47.774,179.215,6.233,149.358
C06829=1133.546,-36.652,-47.786,179.217,6.234,149.358
C06830=1133.541,-36.403,-47.797,179.220,6.234,149.357
C06831=1133.535,-36.153,-47.808,179.223,6.236,149.357
C06832=1133.530,-35.904,-47.820,179.225,6.237,149.356
C06833=1133.525,-35.654,-47.832,179.227,6.237,149.356
C06834=1133.520,-35.404,-47.843,179.230,6.238,149.355
C06835=1133.515,-35.154,-47.855,179.232,6.238,149.355
C06836=1133.509,-34.905,-47.866,179.234,6.239,149.354
C06837=1133.504,-34.655,-47.877,179.237,6.240,149.353
C06838=1133.498,-34.406,-47.889,179.239,6.240,149.353
C06839=1133.494,-34.156,-47.901,179.241,6.241,149.353
C06840=1133.488,-33.906,-47.913,179.244,6.242,149.352
C06841=1133.482,-33.657,-47.924,179.246,6.242,149.351
C06842=1133.478,-33.407,-47.935,179.248,6.243,149.351
C06843=1133.472,-33.157,-47.947,179.250,6.244,149.350
C06844=1133.468,-32.908,-47.959,179.253,6.244,149.350
C06845=1133.462,-32.658,-47.970,179.255,6.245,149.349
C06846=1133.457,-32.408,-47.982,179.257,6.246,149.349
C06847=1133.451,-32.159,-47.993,179.260,6.246,149.348
C06848=1133.446,-31.909,-48.005,179.262,6.247,149.348
C06849=1133.441,-31.659,-48.017,179.265,6.248,149.347
C06850=1133.436,-31.410,-48.029,179.267,6.248,149.346
C06851=1133.431,-31.160,-48.041,179.269,6.249,149.346
C06852=1133.425,-30.910,-48.053,179.272,6.250,149.345
C06853=1133.421,-30.660,-48.064,179.274,6.251,149.345
C06854=1133.415,-30.411,-48.076,179.276,6.251,149.344
C06855=1133.409,-30.161,-48.087,179.279,6.252,149.344
C06856=1133.404,-29.912,-48.099,179.281,6.253,149.343
C06857=1133.399,-29.662,-48.111,179.283,6.253,149.343
C06858=1133.394,-29.412,-48.123,179.286,6.254,149.342
C06859=1133.389,-29.163,-48.135,179.288,6.255,149.342
C06860=1133.384,-28.913,-48.146,179.290,6.255,149.341
C06861=1133.378,-28.663,-48.158,179.293,6.256,149.341
C06862=1133.374,-28.413,-48.170,179.295,6.256,149.340
C06863=1133.369,-28.164,-48.182,179.298,6.258,149.340
C06864=1133.362,-27.915,-48.194,179.300,6.258,149.339
C06865=1133.357,-27.665,-48.206,179.302,6.259,149.338
C06866=1133.352,-27.415,-48.217,179.305,6.260,149.338
C06867=1133.347,-27.165,-48.229,179.307,6.260,149.337
C06868=1133.342,-26.916,-48.241,179.310,6.261,149.337
C06869=1133.336,-26.666,-48.253,179.312,6.262,149.336
C06870=1133.332,-26.416,-48.265,179.314,6.262,149.336
C06871=1133.326,-26.166,-48.276,179.317,6.263,149.335
C06872=1133.321,-25.917,-48.289,179.319,6.264,149.335
C06873=1133.316,-25.667,-48.301,179.321,6.265,149.334
C06874=1133.311,-25.417,-48.312,179.324,6.265,149.333
C06875=1133.305,-25.147,-48.326,179.326,6.266,149.333
C06876=1133.299,-24.877,-48.338,179.329,6.267,149.332
C06877=1133.294,-24.607,-48.351,179.331,6.268,149.332
C06878=1133.288,-24.337,-48.364,179.334,6.268,149.331
C06879=1133.283,-24.088,-48.377,179.336,6.269,149.331
C06880=1133.277,-23.838,-48.388,179.338,6.270,149.330
C06881=1133.272,-23.588,-48.400,179.341,6.270,149.329
C06882=1133.267,-23.339,-48.412,179.344,6.272,149.329
C06883=1133.262,-23.089,-48.424,179.346,6.273,149.329
C06884=1133.257,-22.840,-48.437,179.349,6.273,149.328
C06885=1133.251,-22.590,-48.449,179.351,6.274,149.327
C06886=1133.246,-22.340,-48.461,179.353,6.275,149.327
C06887=1133.241,-22.090,-48.473,179.356,6.275,149.326
C06888=1133.235,-21.841,-48.485,179.358,6.276,149.326
C06889=1133.231,-21.592,-48.497,179.360,6.277,149.325
C06890=1133.226,-21.342,-48.509,179.363,6.277,149.325
C06891=1133.220,-21.092,-48.521,179.365,6.278,149.324
C06892=1133.215,-20.842,-48.533,179.368,6.279,149.324
C06893=1133.210,-20.592,-48.545,179.370,6.280,149.323
C06894=1133.205,-20.343,-48.558,179.372,6.281,149.322
C06895=1133.199,-20.093,-48.570,179.375,6.281,149.322
C06896=1133.194,-19.844,-48.582,179.377,6.282,149.322
C06897=1133.189,-19.594,-48.594,179.379,6.283,149.321
C06898=1133.184,-19.344,-48.607,179.382,6.283,149.320
C06899=1133.179,-19.094,-48.619,179.384,6.284,149.320
C06900=1133.174,-18.845,-48.632,179.386,6.285,149.319
C06901=1133.168,-18.595,-48.644,179.389,6.286,149.319
C06902=1133.164,-18.346,-48.656,179.391,6.287,149.318
C06903=1133.158,-18.096,-48.668,179.394,6.287,149.318
C06904=1133.153,-17.846,-48.680,179.396,6.288,149.317
C06905=1133.148,-17.596,-48.692,179.398,6.289,149.317
C06906=1133.143,-17.347,-48.705,179.401,6.289,149.316
C06907=1133.137,-17.097,-48.717,179.403,6.290,149.315
C06908=1133.132,-16.848,-48.729,179.405,6.291,149.315
C06909=1133.127,-16.599,-48.742,179.408,6.292,149.314
C06910=1133.121,-16.349,-48.754,179.411,6.293,149.314
C06911=1133.117,-16.099,-48.767,179.413,6.294,149.313
C06912=1133.112,-15.849,-48.778,179.415,6.294,149.313
C06913=1133.106,-15.599,-48.791,179.418,6.295,149.312
C06914=1133.101,-15.350,-48.804,179.420,6.296,149.312
C06915=1133.096,-15.100,-48.816,179.422,6.296,149.311
C06916=1133.091,-14.851,-48.828,179.425,6.297,149.311
C06917=1133.085,-14.601,-48.840,179.428,6.298,149.310
C06918=1133.079,-14.351,-48.853,179.430,6.299,149.310
C06919=1133.074,-14.102,-48.866,179.433,6.300,149.309
C06920=1133.069,-13.851,-48.878,179.435,6.300,149.308
C06921=1133.064,-13.602,-48.891,179.437,6.301,149.308
C06922=1133.059,-13.353,-48.903,179.440,6.302,149.307
C06923=1133.054,-13.103,-48.916,179.442,6.302,149.307
C06924=1133.049,-12.853,-48.928,179.445,6.304,149.306
C06925=1133.044,-12.604,-48.940,179.447,6.304,149.306
C06926=1133.039,-12.354,-48.953,179.449,6.305,149.305
C06927=1133.034,-12.104,-48.965,179.452,6.306,149.305
C06928=1133.028,-11.855,-48.978,179.454,6.306,149.304
C06929=1133.023,-11.606,-48.990,179.456,6.307,149.304
C06930=1133.018,-11.356,-49.004,179.459,6.309,149.303
C06931=1133.012,-11.106,-49.015,179.462,6.309,149.302
C06932=1133.008,-10.856,-49.028,179.464,6.310,149.302
C06933=1133.002,-10.607,-49.041,179.466,6.311,149.301
C06934=1132.997,-10.357,-49.054,179.469,6.311,149.301
C06935=1132.992,-10.108,-49.066,179.471,6.312,149.300
C06936=1132.987,-9.858,-49.078,179.474,6.314,149.300
C06937=1132.982,-9.608,-49.091,179.476,6.314,149.299
C06938=1132.976,-9.358,-49.104,179.479,6.315,149.299
C06939=1132.971,-9.109,-49.117,179.481,6.316,149.298
C06940=1132.966,-8.860,-49.129,179.483,6.316,149.298
C06941=1132.962,-8.610,-49.142,179.486,6.318,149.297
C06942=1132.956,-8.360,-49.154,179.489,6.318,149.297
C06943=1132.950,-8.110,-49.168,179.491,6.319,149.296
C06944=1132.945,-7.861,-49.180,179.493,6.320,149.295
C06945=1132.940,-7.612,-49.193,179.496,6.320,149.295
C06946=1132.936,-7.362,-49.206,179.498,6.321,149.294
C06947=1132.930,-7.112,-49.218,179.501,6.322,149.294
C06948=1132.925,-6.863,-49.232,179.503,6.323,149.293
C06949=1132.919,-6.613,-49.244,179.505,6.324,149.293
C06950=1132.915,-6.363,-49.257,179.508,6.324,149.292
C06951=1132.909,-6.113,-49.269,179.510,6.325,149.292
C06952=1132.904,-5.864,-49.282,179.513,6.327,149.291
C06953=1132.898,-5.614,-49.295,179.516,6.327,149.290
C06954=1132.894,-5.364,-49.308,179.518,6.328,149.290
C06955=1132.889,-5.115,-49.320,179.520,6.329,149.290
C06956=1132.883,-4.865,-49.334,179.523,6.329,149.289
C06957=1132.878,-4.615,-49.346,179.525,6.331,149.288
C06958=1132.873,-4.366,-49.359,179.528,6.332,149.288
C06959=1132.867,-4.116,-49.372,179.530,6.332,149.287
C06960=1132.862,-3.867,-49.385,179.532,6.333,149.287
C06961=1132.858,-3.617,-49.398,179.535,6.334,149.286
C06962=1132.853,-3.368,-49.410,179.538,6.335,149.286
C06963=1132.847,-3.118,-49.424,179.540,6.336,149.285
C06964=1132.842,-2.868,-49.437,179.542,6.336,149.285
C06965=1132.837,-2.619,-49.449,179.545,6.337,149.284
C06966=1132.831,-2.369,-49.462,179.548,6.338,149.284
C06967=1132.827,-2.120,-49.476,179.550,6.339,149.283
C06968=1132.822,-1.870,-49.489,179.553,6.340,149.282
C06969=1132.816,-1.621,-49.502,179.555,6.340,149.282
C06970=1132.812,-1.371,-49.515,179.557,6.342,149.281
C06971=1132.806,-1.121,-49.528,179.560,6.342,149.281
C06972=1132.801,-0.872,-49.541,179.562,6.343,149.280
C06973=1132.796,-0.622,-49.554,179.564,6.344,149.280
C06974=1132.790,-0.372,-49.567,179.567,6.346,149.279
C06975=1132.785,-0.123,-49.579,179.570,6.346,149.279
C06976=1132.781,0.127,-49.593,179.572,6.347,149.278
C06977=1132.775,0.376,-49.606,179.574,6.348,149.278
C06978=1132.771,0.626,-49.619,179.577,6.348,149.277
C06979=1132.764,0.895,-49.633,179.580,6.350,149.277
C06980=1132.759,1.165,-49.648,179.582,6.350,149.276
C06981=1132.754,1.435,-49.662,179.585,6.352,149.275
C06982=1132.747,1.704,-49.676,179.588,6.352,149.275
C06983=1132.743,1.954,-49.689,179.590,6.353,149.274
C06984=1132.737,2.203,-49.703,179.593,6.354,149.274
C06985=1132.732,2.452,-49.715,179.595,6.355,149.273
C06986=1132.727,2.703,-49.729,179.598,6.356,149.273
C06987=1132.722,2.952,-49.741,179.600,6.356,149.272
C06988=1132.717,3.202,-49.756,179.603,6.358,149.271
C06989=1132.712,3.451,-49.768,179.605,6.358,149.271
C06990=1132.706,3.701,-49.782,179.607,6.359,149.271
C06991=1132.701,3.951,-49.794,179.611,6.361,149.270
C06992=1132.696,4.200,-49.808,179.613,6.361,149.269
C06993=1132.691,4.450,-49.821,179.615,6.362,149.269
C06994=1132.685,4.699,-49.835,179.618,6.363,149.268
C06995=1132.681,4.949,-49.848,179.620,6.364,149.268
C06996=1132.675,5.198,-49.861,179.623,6.365,149.267
C06997=1132.671,5.448,-49.874,179.625,6.365,149.267
C06998=1132.665,5.697,-49.888,179.627,6.366,149.266
C06999=1132.661,5.947,-49.901,179.630,6.368,149.266
C07000=1132.655,6.197,-49.914,179.633,6.368,149.265
C07001=1132.651,6.446,-49.928,179.635,6.369,149.265
C07002=1132.645,6.696,-49.941,179.638,6.371,149.264
C07003=1132.640,6.945,-49.955,179.640,6.371,149.263
C07004=1132.635,7.195,-49.968,179.643,6.372,149.263
C07005=1132.629,7.445,-49.981,179.645,6.373,149.262
C07006=1132.625,7.694,-49.995,179.648,6.374,149.262
C07007=1132.619,7.944,-50.008,179.650,6.375,149.261
C07008=1132.615,8.193,-50.022,179.652,6.375,149.261
C07009=1132.609,8.443,-50.035,179.656,6.377,149.260
C07010=1132.604,8.692,-50.049,179.658,6.377,149.260
C07011=1132.599,8.942,-50.062,179.660,6.378,149.259
C07012=1132.593,9.192,-50.076,179.663,6.379,149.259
C07013=1132.589,9.441,-50.089,179.665,6.380,149.258
C07014=1132.583,9.691,-50.102,179.668,6.381,149.258
C07015=1132.578,9.941,-50.117,179.670,6.382,149.257
C07016=1132.573,10.190,-50.129,179.673,6.383,149.257
C07017=1132.568,10.440,-50.144,179.675,6.384,149.256
C07018=1132.562,10.689,-50.157,179.678,6.384,149.255
C07019=1132.558,10.939,-50.170,179.681,6.386,149.255
C07020=1132.552,11.189,-50.184,179.683,6.387,149.254
C07021=1132.547,11.438,-50.198,179.686,6.387,149.254
C07022=1132.543,11.687,-50.211,179.688,6.389,149.253
C07023=1132.537,11.937,-50.225,179.690,6.390,149.253
C07024=1132.532,12.186,-50.239,179.693,6.390,149.252
C07025=1132.527,12.436,-50.252,179.696,6.392,149.252
C07026=1132.522,12.686,-50.266,179.698,6.392,149.251
C07027=1132.517,12.935,-50.280,179.700,6.393,149.251
C07028=1132.511,13.185,-50.293,179.704,6.394,149.250
C07029=1132.507,13.434,-50.307,179.706,6.395,149.250
C07030=1132.501,13.684,-50.320,179.708,6.396,149.249
C07031=1132.496,13.934,-50.335,179.711,6.397,149.248
C07032=1132.491,14.183,-50.349,179.713,6.398,149.248
C07033=1132.486,14.433,-50.361,179.715,6.399,149.248
C07034=1132.481,14.682,-50.375,179.719,6.400,149.247
C07035=1132.476,14.932,-50.390,179.721,6.401,149.246
C07036=1132.471,15.182,-50.403,179.723,6.402,149.246
C07037=1132.466,15.431,-50.417,179.726,6.403,149.245
C07038=1132.461,15.681,-50.431,179.728,6.404,149.245
C07039=1132.455,15.930,-50.444,179.731,6.405,149.244
C07040=1132.450,16.180,-50.458,179.734,6.406,149.244
C07041=1132.445,16.430,-50.473,179.736,6.407,149.243
C07042=1132.440,16.678,-50.486,179.738,6.407,149.243
C07043=1132.435,16.929,-50.499,179.741,6.409,149.242
C07044=1132.430,17.178,-50.514,179.744,6.410,149.242
C07045=1132.424,17.427,-50.528,179.746,6.411,149.241
C07046=1132.419,17.677,-50.542,179.749,6.412,149.240
C07047=1132.414,17.927,-50.555,179.751,6.412,149.240
C07048=1132.409,18.176,-50.569,179.754,6.414,149.240
C07049=1132.404,18.426,-50.583,179.757,6.414,149.239
C07050=1132.399,18.676,-50.597,179.759,6.415,149.238
C07051=1132.394,18.925,-50.611,179.762,6.417,149.238
C07052=1132.389,19.174,-50.626,179.764,6.417,149.237
C07053=1132.384,19.425,-50.639,179.767,6.419,149.237
C07054=1132.378,19.674,-50.653,179.769,6.420,149.236
C07055=1132.373,19.923,-50.667,179.771,6.420,149.236
C07056=1132.368,20.173,-50.682,179.775,6.422,149.235
C07057=1132.364,20.422,-50.695,179.777,6.423,149.235
C07058=1132.358,20.671,-50.709,179.779,6.423,149.234
C07059=1132.353,20.921,-50.723,179.782,6.425,149.234
C07060=1132.349,21.171,-50.738,179.784,6.425,149.233
C07061=1132.343,21.420,-50.751,179.787,6.427,149.233
C07062=1132.338,21.670,-50.765,179.790,6.427,149.232
C07063=1132.333,21.920,-50.779,179.792,6.428,149.232
C07064=1132.328,22.170,-50.794,179.795,6.430,149.231
C07065=1132.322,22.419,-50.808,179.797,6.430,149.230
C07066=1132.317,22.668,-50.822,179.800,6.432,149.230
C07067=1132.312,22.918,-50.836,179.802,6.433,149.229
C07068=1132.307,23.168,-50.850,179.805,6.433,149.229
C07069=1132.302,23.417,-50.864,179.808,6.435,149.228
C07070=1132.297,23.666,-50.879,179.810,6.436,149.228
C07071=1132.292,23.916,-50.893,179.813,6.437,149.227
C07072=1132.287,24.166,-50.907,179.815,6.438,149.227
C07073=1132.281,24.415,-50.921,179.818,6.438,149.226
C07074=1132.276,24.665,-50.935,179.821,6.440,149.226
C07075=1132.272,24.914,-50.950,179.823,6.440,149.225
C07076=1132.267,25.164,-50.964,179.826,6.442,149.225
C07077=1132.262,25.414,-50.978,179.828,6.443,149.224
C07078=1132.256,25.663,-50.992,179.831,6.443,149.224
C07079=1132.251,25.912,-51.006,179.833,6.445,149.223
C07080=1132.246,26.162,-51.021,179.836,6.446,149.223
C07081=1132.241,26.411,-51.036,179.839,6.447,149.222
C07082=1132.237,26.661,-51.050,179.841,6.448,149.222
C07083=1132.231,26.930,-51.065,179.844,6.449,149.221
C07084=1132.225,27.199,-51.081,179.846,6.450,149.220
C07085=1132.219,27.468,-51.096,179.849,6.451,149.220
C07086=1132.214,27.737,-51.112,179.852,6.453,149.219
C07087=1132.209,27.987,-51.126,179.855,6.454,149.219
C07088=1132.204,28.236,-51.140,179.858,6.455,149.218
C07089=1132.200,28.485,-51.155,179.860,6.456,149.218
C07090=1132.194,28.734,-51.169,179.862,6.456,149.217
C07091=1132.188,28.985,-51.184,179.865,6.458,149.217
C07092=1132.183,29.234,-51.198,179.868,6.458,149.216
C07093=1132.178,29.484,-51.213,179.870,6.460,149.216
C07094=1132.174,29.733,-51.228,179.872,6.461,149.215
C07095=1132.169,29.983,-51.242,179.876,6.462,149.214
C07096=1132.164,30.232,-51.256,179.878,6.463,149.214
C07097=1132.158,30.482,-51.271,179.881,6.465,149.214
C07098=1132.153,30.731,-51.286,179.883,6.465,149.213
C07099=1132.148,30.981,-51.300,179.885,6.466,149.212
C07100=1132.143,31.230,-51.314,179.888,6.467,149.212
C07101=1132.138,31.480,-51.328,179.891,6.468,149.211
C07102=1132.133,31.729,-51.343,179.894,6.469,149.211
C07103=1132.128,31.979,-51.358,179.896,6.470,149.210
C07104=1132.123,32.229,-51.373,179.899,6.472,149.210
C07105=1132.118,32.478,-51.388,179.901,6.472,149.209
C07106=1132.113,32.728,-51.402,179.904,6.474,149.209
C07107=1132.107,32.978,-51.417,179.906,6.475,149.208
C07108=1132.103,33.227,-51.432,179.909,6.476,149.208
C07109=1132.098,33.476,-51.446,179.912,6.477,149.207
C07110=1132.092,33.725,-51.460,179.914,6.478,149.207
C07111=1132.087,33.975,-51.475,179.917,6.479,149.206
C07112=1132.082,34.225,-51.490,179.920,6.481,149.206
C07113=1132.077,34.474,-51.505,179.922,6.481,149.205
C07114=1132.072,34.723,-51.519,179.925,6.483,149.205
C07115=1132.067,34.973,-51.534,179.927,6.483,149.204
C07116=1132.062,35.222,-51.549,179.930,6.485,149.204
C07117=1132.057,35.472,-51.563,179.932,6.486,149.203
C07118=1132.052,35.722,-51.579,179.935,6.486,149.203
C07119=1132.047,35.971,-51.593,179.938,6.488,149.202
C07120=1132.042,36.220,-51.608,179.940,6.489,149.202
C07121=1132.036,36.470,-51.623,179.943,6.490,149.201
C07122=1132.032,36.720,-51.638,179.945,6.491,149.200
C07123=1132.027,36.969,-51.652,179.948,6.492,149.200
C07124=1132.021,37.219,-51.668,179.951,6.493,149.199
C07125=1132.016,37.468,-51.682,179.953,6.494,149.199
C07126=1132.012,37.717,-51.697,179.956,6.495,149.198
C07127=1132.006,37.967,-51.712,179.958,6.497,149.198
C07128=1132.001,38.217,-51.727,179.962,6.498,149.197
C07129=1131.996,38.467,-51.742,179.964,6.499,149.197
C07130=1131.991,38.716,-51.757,179.967,6.501,149.196
C07131=1131.986,38.965,-51.771,179.969,6.501,149.196
C07132=1131.981,39.215,-51.787,179.972,6.503,149.195
C07133=1131.976,39.464,-51.802,179.974,6.504,149.195
C07134=1131.970,39.714,-51.816,179.977,6.505,149.194
C07135=1131.966,39.963,-51.831,179.980,6.506,149.194
C07136=1131.961,40.213,-51.846,179.982,6.507,149.193
C07137=1131.955,40.462,-51.861,179.984,6.508,149.193
C07138=1131.951,40.711,-51.876,179.988,6.509,149.192
C07139=1131.945,40.961,-51.891,179.990,6.510,149.192
C07140=1131.941,41.211,-51.907,179.993,6.512,149.191
C07141=1131.936,41.460,-51.922,179.995,6.513,149.191
C07142=1131.931,41.710,-51.936,179.998,6.514,149.190
C07143=1131.925,41.960,-51.952,-180.000,6.515,149.190
C07144=1131.921,42.209,-51.967,-179.997,6.516,149.189
C07145=1131.915,42.459,-51.982,-179.994,6.517,149.189
C07146=1131.910,42.708,-51.997,-179.992,6.518,149.188
C07147=1131.905,42.957,-52.012,-179.989,6.520,149.188
C07148=1131.900,43.206,-52.027,-179.987,6.521,149.187
C07149=1131.895,43.456,-52.042,-179.983,6.522,149.187
C07150=1131.890,43.706,-52.058,-179.981,6.523,149.186
C07151=1131.885,43.955,-52.073,-179.978,6.524,149.186
C07152=1131.880,44.205,-52.088,-179.976,6.525,149.185
C07153=1131.875,44.455,-52.103,-179.973,6.527,149.185
C07154=1131.870,44.704,-52.118,-179.971,6.527,149.184
C07155=1131.865,44.953,-52.134,-179.968,6.529,149.184
C07156=1131.860,45.202,-52.149,-179.965,6.530,149.183
C07157=1131.855,45.452,-52.164,-179.963,6.531,149.183
C07158=1131.850,45.702,-52.180,-179.960,6.533,149.182
C07159=1131.845,45.951,-52.194,-179.957,6.533,149.181
C07160=1131.840,46.201,-52.210,-179.955,6.535,149.181
C07161=1131.835,46.450,-52.225,-179.952,6.536,149.181
C07162=1131.830,46.699,-52.241,-179.950,6.537,149.180
C07163=1131.824,46.949,-52.256,-179.946,6.538,149.179
C07164=1131.820,47.198,-52.272,-179.944,6.539,149.179
C07165=1131.815,47.448,-52.287,-179.941,6.541,149.178
C07166=1131.810,47.698,-52.301,-179.939,6.541,149.178
C07167=1131.804,47.947,-52.317,-179.936,6.543,149.177
C07168=1131.799,48.196,-52.333,-179.934,6.544,149.177
C07169=1131.795,48.446,-52.348,-179.931,6.545,149.176
C07170=1131.790,48.696,-52.364,-179.928,6.547,149.176
C07171=1131.784,48.945,-52.379,-179.926,6.548,149.175
C07172=1131.779,49.194,-52.394,-179.923,6.549,149.175
C07173=1131.775,49.444,-52.410,-179.921,6.550,149.174
C07174=1131.769,49.694,-52.426,-179.918,6.551,149.174
C07175=1131.765,49.943,-52.441,-179.915,6.553,149.173
C07176=1131.759,50.192,-52.456,-179.913,6.554,149.173
C07177=1131.754,50.441,-52.472,-179.909,6.555,149.172
C07178=1131.750,50.691,-52.487,-179.907,6.556,149.172
C07179=1131.744,50.941,-52.503,-179.905,6.557,149.171
C07180=1131.739,51.190,-52.518,-179.902,6.559,149.171
C07181=1131.734,51.440,-52.534,-179.899,6.560,149.170
C07182=1131.730,51.689,-52.549,-179.896,6.561,149.170
C07183=1131.724,51.939,-52.565,-179.894,6.562,149.169
C07184=1131.719,52.187,-52.581,-179.891,6.564,149.169
C07185=1131.714,52.438,-52.597,-179.888,6.565,149.168
C07186=1131.710,52.687,-52.612,-179.886,6.566,149.168
C07187=1131.704,52.955,-52.629,-179.883,6.567,149.167
C07188=1131.698,53.224,-52.646,-179.880,6.569,149.167
C07189=1131.693,53.493,-52.663,-179.877,6.570,149.166
C07190=1131.687,53.761,-52.680,-179.874,6.571,149.166
C07191=1131.682,54.011,-52.696,-179.872,6.572,149.165
C07192=1131.678,54.260,-52.711,-179.869,6.574,149.165
C07193=1131.673,54.509,-52.727,-179.867,6.575,149.164
C07194=1131.668,54.759,-52.743,-179.864,6.576,149.164
C07195=1131.663,55.009,-52.758,-179.861,6.578,149.163
C07196=1131.657,55.258,-52.774,-179.859,6.579,149.163
C07197=1131.652,55.508,-52.790,-179.856,6.580,149.162
C07198=1131.647,55.757,-52.806,-179.853,6.581,149.162
C07199=1131.643,56.006,-52.821,-179.851,6.582,149.161
C07200=1131.638,56.256,-52.837,-179.848,6.584,149.161
C07201=1131.632,56.506,-52.853,-179.845,6.585,149.160
C07202=1131.627,56.754,-52.869,-179.842,6.586,149.160
C07203=1131.623,57.004,-52.885,-179.840,6.588,149.159
C07204=1131.617,57.254,-52.901,-179.838,6.588,149.159
C07205=1131.612,57.503,-52.917,-179.834,6.590,149.158
C07206=1131.607,57.753,-52.933,-179.832,6.591,149.158
C07207=1131.602,58.002,-52.948,-179.829,6.592,149.157
C07208=1131.598,58.252,-52.964,-179.827,6.594,149.157
C07209=1131.593,58.501,-52.980,-179.823,6.595,149.156
C07210=1131.587,58.750,-52.996,-179.821,6.596,149.156
C07211=1131.583,59.000,-53.012,-179.819,6.598,149.155
C07212=1131.578,59.249,-53.028,-179.816,6.599,149.155
C07213=1131.573,59.499,-53.044,-179.813,6.600,149.154
C07214=1131.568,59.748,-53.060,-179.810,6.601,149.154
C07215=1131.562,59.997,-53.076,-179.808,6.603,149.153
C07216=1131.557,60.247,-53.092,-179.805,6.604,149.153
C07217=1131.552,60.496,-53.108,-179.803,6.605,149.152
C07218=1131.548,60.746,-53.124,-179.799,6.607,149.152
C07219=1131.543,60.995,-53.140,-179.797,6.607,149.151
C07220=1131.538,61.245,-53.156,-179.795,6.609,149.151
C07221=1131.533,61.494,-53.173,-179.792,6.611,149.150
C07222=1131.527,61.743,-53.188,-179.789,6.611,149.150
C07223=1131.523,61.993,-53.205,-179.786,6.613,149.149
C07224=1131.517,62.242,-53.220,-179.784,6.614,149.149
C07225=1131.513,62.492,-53.237,-179.781,6.616,149.148
C07226=1131.508,62.741,-53.253,-179.778,6.617,149.148
C07227=1131.503,62.991,-53.269,-179.775,6.618,149.147
C07228=1131.498,63.240,-53.285,-179.773,6.620,149.147
C07229=1131.493,63.489,-53.302,-179.771,6.621,149.146
C07230=1131.487,63.739,-53.318,-179.767,6.622,149.146
C07231=1131.483,63.989,-53.334,-179.765,6.624,149.145
C07232=1131.477,64.238,-53.350,-179.762,6.624,149.145
C07233=1131.473,64.488,-53.367,-179.760,6.626,149.144
C07234=1131.468,64.736,-53.383,-179.756,6.627,149.144
C07235=1131.463,64.986,-53.399,-179.754,6.629,149.143
C07236=1131.458,65.235,-53.415,-179.752,6.630,149.143
C07237=1131.453,65.485,-53.431,-179.749,6.631,149.142
C07238=1131.448,65.734,-53.447,-179.746,6.633,149.142
C07239=1131.443,65.984,-53.464,-179.743,6.634,149.141
C07240=1131.437,66.233,-53.480,-179.741,6.635,149.141
C07241=1131.433,66.483,-53.497,-179.738,6.637,149.140
C07242=1131.428,66.732,-53.513,-179.735,6.639,149.140
C07243=1131.423,66.982,-53.529,-179.732,6.639,149.139
C07244=1131.418,67.231,-53.546,-179.730,6.641,149.139
C07245=1131.413,67.480,-53.562,-179.727,6.642,149.139
C07246=1131.408,67.730,-53.580,-179.725,6.643,149.138
C07247=1131.403,67.979,-53.595,-179.722,6.645,149.138
C07248=1131.398,68.229,-53.612,-179.719,6.646,149.137
C07249=1131.393,68.477,-53.628,-179.716,6.648,149.137
C07250=1131.388,68.727,-53.644,-179.714,6.649,149.136
C07251=1131.383,68.977,-53.661,-179.711,6.650,149.136
C07252=1131.378,69.226,-53.678,-179.708,6.651,149.135
C07253=1131.374,69.476,-53.694,-179.705,6.653,149.135
C07254=1131.369,69.724,-53.711,-179.703,6.654,149.134
C07255=1131.363,69.975,-53.727,-179.700,6.656,149.134
C07256=1131.359,70.224,-53.744,-179.698,6.657,149.133
C07257=1131.354,70.473,-53.760,-179.694,6.658,149.133
C07258=1131.349,70.722,-53.777,-179.692,6.659,149.132
C07259=1131.343,70.972,-53.794,-179.689,6.661,149.132
C07260=1131.339,71.221,-53.810,-179.687,6.663,149.131
C07261=1131.334,71.471,-53.826,-179.684,6.664,149.131
C07262=1131.328,71.720,-53.843,-179.681,6.665,149.130
C07263=1131.324,71.970,-53.860,-179.678,6.666,149.130
C07264=1131.319,72.219,-53.877,-179.676,6.668,149.129
C07265=1131.313,72.468,-53.893,-179.673,6.670,149.129
C07266=1131.309,72.718,-53.910,-179.671,6.670,149.128
C07267=1131.304,72.967,-53.926,-179.668,6.672,149.128
C07268=1131.299,73.216,-53.944,-179.665,6.673,149.127
C07269=1131.294,73.466,-53.960,-179.662,6.675,149.127
C07270=1131.290,73.715,-53.977,-179.659,6.677,149.127
C07271=1131.284,73.964,-53.994,-179.657,6.678,149.126
C07272=1131.279,74.214,-54.011,-179.654,6.679,149.125
C07273=1131.275,74.463,-54.027,-179.651,6.680,149.125
C07274=1131.269,74.713,-54.044,-179.648,6.682,149.125
C07275=1131.265,74.962,-54.061,-179.646,6.683,149.124
C07276=1131.259,75.212,-54.078,-179.644,6.685,149.124
C07277=1131.254,75.461,-54.094,-179.640,6.686,149.123
C07278=1131.250,75.710,-54.111,-179.638,6.688,149.123
C07279=1131.245,75.960,-54.128,-179.635,6.689,149.122
C07280=1131.239,76.209,-54.145,-179.633,6.690,149.122
C07281=1131.234,76.458,-54.162,-179.630,6.692,149.121
C07282=1131.230,76.708,-54.179,-179.627,6.693,149.121
C07283=1131.225,76.958,-54.196,-179.624,6.695,149.120
C07284=1131.219,77.207,-54.212,-179.621,6.696,149.120
C07285=1131.214,77.456,-54.229,-179.619,6.697,149.119
C07286=1131.210,77.705,-54.247,-179.616,6.699,149.119
C07287=1131.206,77.955,-54.263,-179.613,6.700,149.118
C07288=1131.200,78.204,-54.280,-179.610,6.702,149.118
C07289=1131.195,78.453,-54.297,-179.608,6.703,149.117
C07290=1131.190,78.703,-54.314,-179.605,6.705,149.117
C07291=1131.168,79.846,-54.396,179.909,7.658,149.472
C07292=1131.163,80.095,-54.414,179.910,7.662,149.472
C07293=1131.158,80.345,-54.430,179.911,7.665,149.473
C07294=1131.153,80.594,-54.448,179.912,7.670,149.473
C07295=1131.147,80.843,-54.465,179.913,7.673,149.474
C07296=1131.143,81.092,-54.483,179.914,7.677,149.474
C07297=1131.138,81.342,-54.500,179.916,7.681,149.475
C07298=1131.133,81.591,-54.518,179.917,7.684,149.475
C07299=1131.129,81.840,-54.534,179.918,7.688,149.476
C07300=1131.123,82.090,-54.552,179.919,7.691,149.476
C07301=1131.119,82.339,-54.570,179.920,7.696,149.477
C07302=1131.114,82.589,-54.586,179.922,7.700,149.477
C07303=1131.109,82.838,-54.604,179.922,7.703,149.478
C07304=1131.103,83.087,-54.621,179.924,7.707,149.479
